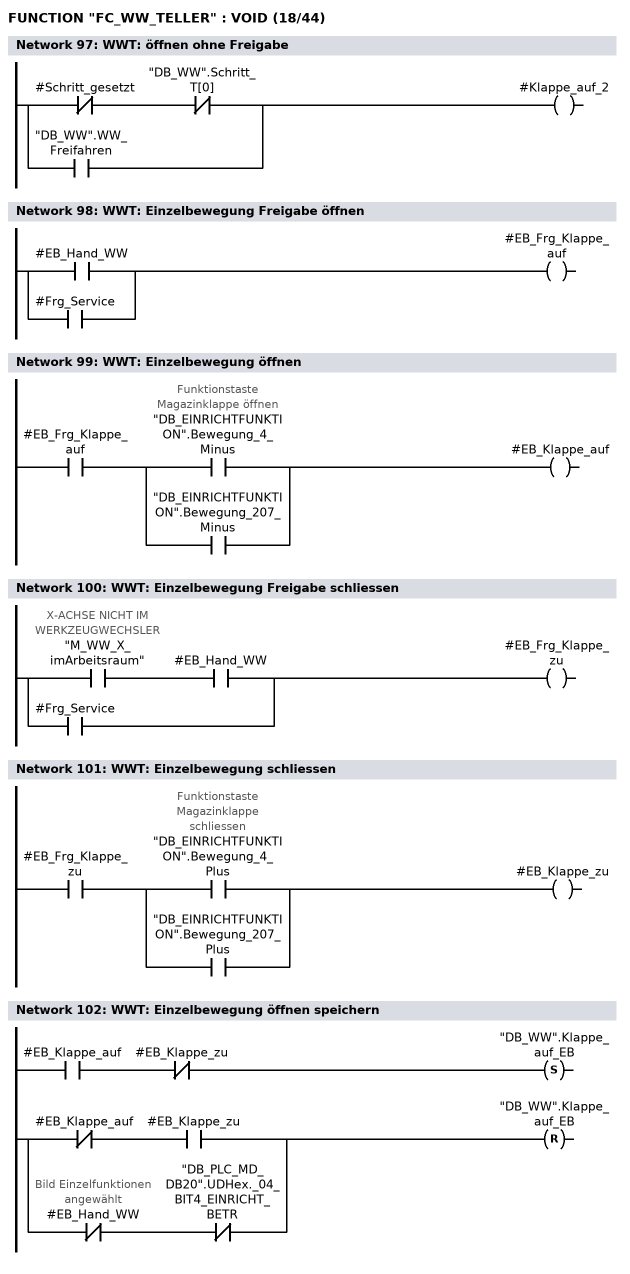

      UN    #Schritt_gesetzt;
      UN    "DB_WW".Schritt_T[0];
      O     "DB_WW".WW_Freifahren;
      =     #Klappe_auf_2;

NETWORK
TITLE =WWT: Einzelbewegung Freigabe öffnen

      O     #EB_Hand_WW;
      O     #Frg_Service;
      =     #EB_Frg_Klappe_auf;

NETWORK
TITLE =WWT: Einzelbewegung öffnen

      U     #EB_Frg_Klappe_auf;
      U(    ;
      O     "DB_EINRICHTFUNKTION".Bewegung_4_Minus; // Funktionstaste Magazinklappe öffnen
      O     "DB_EINRICHTFUNKTION".Bewegung_207_Minus;
      )     ;
      =     #EB_Klappe_auf;

NETWORK
TITLE =WWT: Einzelbewegung Freigabe schliessen

      U     "M_WW_X_imArbeitsraum"; // X-ACHSE NICHT IM WERKZEUGWECHSLER
      U     #EB_Hand_WW;
      O     #Frg_Service;
      =     #EB_Frg_Klappe_zu;

NETWORK
TITLE =WWT: Einzelbewegung schliessen

      U     #EB_Frg_Klappe_zu;
      U(    ;
      O     "DB_EINRICHTFUNKTION".Bewegung_4_Plus; // Funktionstaste Magazinklappe schliessen
      O     "DB_EINRICHTFUNKTION".Bewegung_207_Plus;
      )     ;
      =     #EB_Klappe_zu;

NETWORK
TITLE =WWT: Einzelbewegung öffnen speichern

      U     #EB_Klappe_auf;
      UN    #EB_Klappe_zu;
      S     "DB_WW".Klappe_auf_EB;

      U(    ;
      UN    #EB_Klappe_auf;
      U     #EB_Klappe_zu;
      O     ;
      UN    #EB_Hand_WW; // Bild Einzelfunktionen angewählt
      UN    "DB_PLC_MD_DB20".UDHex._04_BIT4_EINRICHT_BETR;
      )     ;
      R     "DB_WW".Klappe_auf_EB;
      NOP   0;

NETWORK
TITLE =WWT: Einzelbewegung schliessen speichern
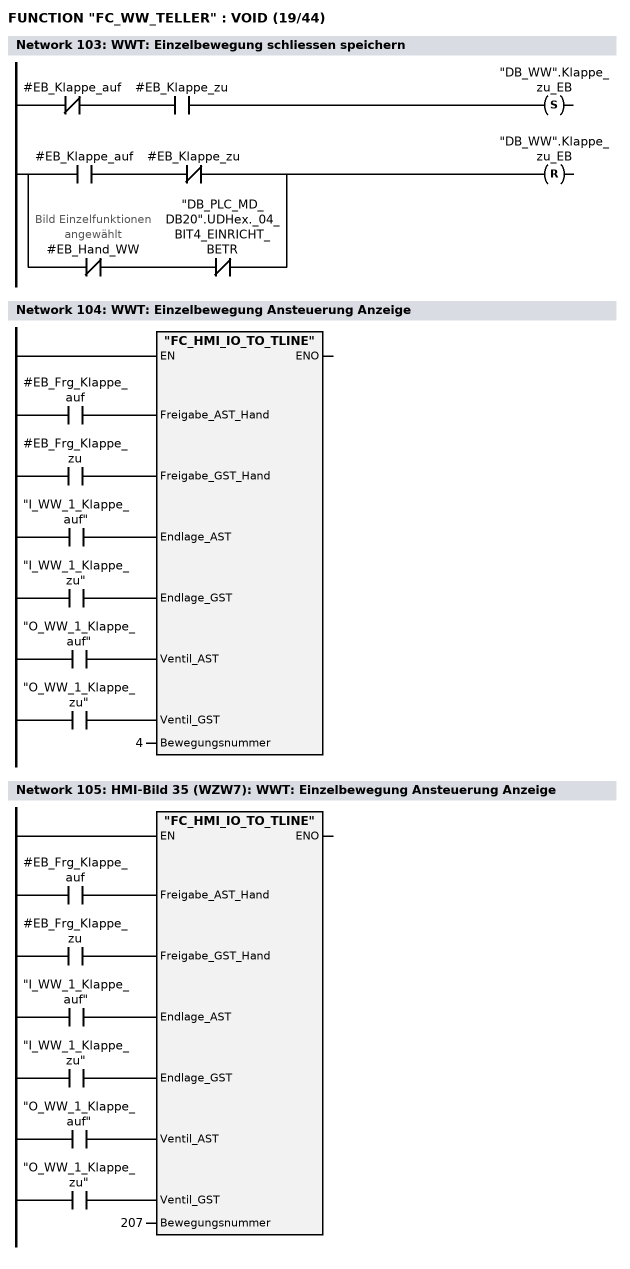

      UN    #EB_Klappe_auf;
      U     #EB_Klappe_zu;
      S     "DB_WW".Klappe_zu_EB;

      U(    ;
      U     #EB_Klappe_auf;
      UN    #EB_Klappe_zu;
      O     ;
      UN    #EB_Hand_WW; // Bild Einzelfunktionen angewählt
      UN    "DB_PLC_MD_DB20".UDHex._04_BIT4_EINRICHT_BETR;
      )     ;
      R     "DB_WW".Klappe_zu_EB;
      NOP   0;

NETWORK
TITLE =WWT: Einzelbewegung Ansteuerung Anzeige

      U     #EB_Frg_Klappe_auf;
      =     L     24.0;
      BLD   103;
      U     #EB_Frg_Klappe_zu;
      =     L     24.1;
      BLD   103;
      U     "I_WW_1_Klappe_auf";
      =     L     24.2;
      BLD   103;
      U     "I_WW_1_Klappe_zu";
      =     L     24.3;
      BLD   103;
      U     "O_WW_1_Klappe_auf";
      =     L     24.4;
      BLD   103;
      U     "O_WW_1_Klappe_zu";
      =     L     24.5;
      BLD   103;
      CALL "FC_HMI_IO_TO_TLINE" (
           Freigabe_AST_Hand        := L     24.0,
           Freigabe_GST_Hand        := L     24.1,
           Endlage_AST              := L     24.2,
           Endlage_GST              := L     24.3,
           Ventil_AST               := L     24.4,
           Ventil_GST               := L     24.5,
           Bewegungsnummer          := 4);
      NOP   0;
NETWORK
TITLE =HMI-Bild 35 (WZW7): WWT: Einzelbewegung Ansteuerung Anzeige

      U     #EB_Frg_Klappe_auf;
      =     L     24.0;
      BLD   103;
      U     #EB_Frg_Klappe_zu;
      =     L     24.1;
      BLD   103;
      U     "I_WW_1_Klappe_auf";
      =     L     24.2;
      BLD   103;
      U     "I_WW_1_Klappe_zu";
      =     L     24.3;
      BLD   103;
      U     "O_WW_1_Klappe_auf";
      =     L     24.4;
      BLD   103;
      U     "O_WW_1_Klappe_zu";
      =     L     24.5;
      BLD   103;
      CALL "FC_HMI_IO_TO_TLINE" (
           Freigabe_AST_Hand        := L     24.0,
           Freigabe_GST_Hand        := L     24.1,
           Endlage_AST              := L     24.2,
           Endlage_GST              := L     24.3,
           Ventil_AST               := L     24.4,
           Ventil_GST               := L     24.5,
           Bewegungsnummer          := 207);
      NOP   0;
NETWORK
TITLE =WWT: Ausgang öffnen
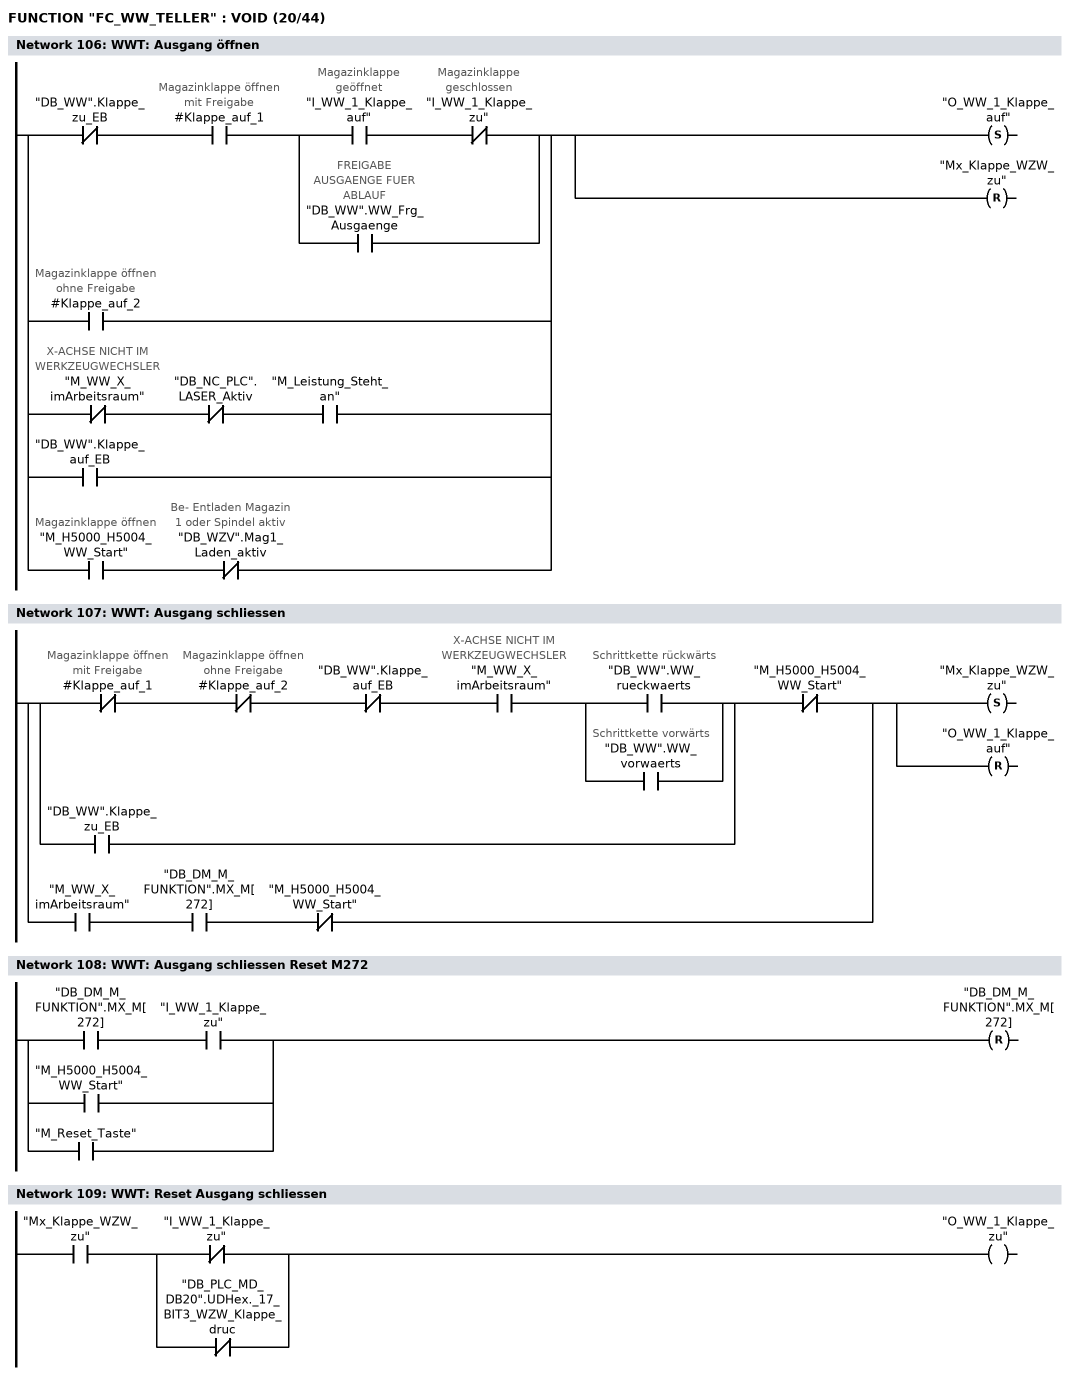

      UN    "DB_WW".Klappe_zu_EB;
      U     #Klappe_auf_1; // Magazinklappe öffnen mit Freigabe
      U(    ;
      U     "I_WW_1_Klappe_auf"; // Magazinklappe geöffnet
      UN    "I_WW_1_Klappe_zu"; // Magazinklappe geschlossen
      O     "DB_WW".WW_Frg_Ausgaenge; // FREIGABE AUSGAENGE FUER ABLAUF
      )     ;
      O     #Klappe_auf_2; // Magazinklappe öffnen ohne Freigabe
      O     ;
      UN    "M_WW_X_imArbeitsraum"; // X-ACHSE NICHT IM WERKZEUGWECHSLER
      UN    "DB_NC_PLC".LASER_Aktiv;
      U     "M_Leistung_Steht_an";
      O     "DB_WW".Klappe_auf_EB;
      O     ;
      U     "M_H5000_H5004_WW_Start"; // Magazinklappe öffnen
      UN    "DB_WZV".Mag1_Laden_aktiv; // Be- Entladen Magazin 1 oder Spindel aktiv
      S     "O_WW_1_Klappe_auf";

      R     "Mx_Klappe_WZW_zu";
NETWORK
TITLE =WWT: Ausgang schliessen

      U(    ;
      UN    #Klappe_auf_1; // Magazinklappe öffnen mit Freigabe
      UN    #Klappe_auf_2; // Magazinklappe öffnen ohne Freigabe
      UN    "DB_WW".Klappe_auf_EB;
      U     "M_WW_X_imArbeitsraum"; // X-ACHSE NICHT IM WERKZEUGWECHSLER
//      U     "I_WW_1_Klappe_zu"
      U(    ;
      O     "DB_WW".WW_rueckwaerts; // Schrittkette rückwärts
      O     "DB_WW".WW_vorwaerts; // Schrittkette vorwärts
      )     ;
      O     "DB_WW".Klappe_zu_EB;
      )     ;
      UN    "M_H5000_H5004_WW_Start";
      O     ;
      U     "M_WW_X_imArbeitsraum";
      U     "DB_DM_M_FUNKTION".MX_M[272];
      UN    "M_H5000_H5004_WW_Start";
      S     "Mx_Klappe_WZW_zu";
      R     "O_WW_1_Klappe_auf";

NETWORK
TITLE =WWT: Ausgang schliessen Reset M272

      U     "DB_DM_M_FUNKTION".MX_M[272];
      U     "I_WW_1_Klappe_zu";
      O     "M_H5000_H5004_WW_Start";
      O     "M_Reset_Taste";
      R     "DB_DM_M_FUNKTION".MX_M[272];

NETWORK
TITLE =WWT: Reset Ausgang schliessen

      U     "Mx_Klappe_WZW_zu";
      U(    ;
      ON    "I_WW_1_Klappe_zu";
      ON    "DB_PLC_MD_DB20".UDHex._17_BIT3_WZW_Klappe_druc;
      )     ;
      =     "O_WW_1_Klappe_zu";

NETWORK
TITLE =========== Werkzeug in / aus Spindel ===============



NETWORK
TITLE =WZHUB: BEFEHL FAHRE auf AUSFAHRPOSITION
// AUS DEN SCHRITTMERKERN WERDEN VERSCHIEDENE BEFEHLE ERZEUGT, DIE
// WIEDERUM VERSCHIEDENE AKTION AUSLOESEN.
//
// BEFEHL FAHRE Z-Achse auf AUSFAHRPOSITION
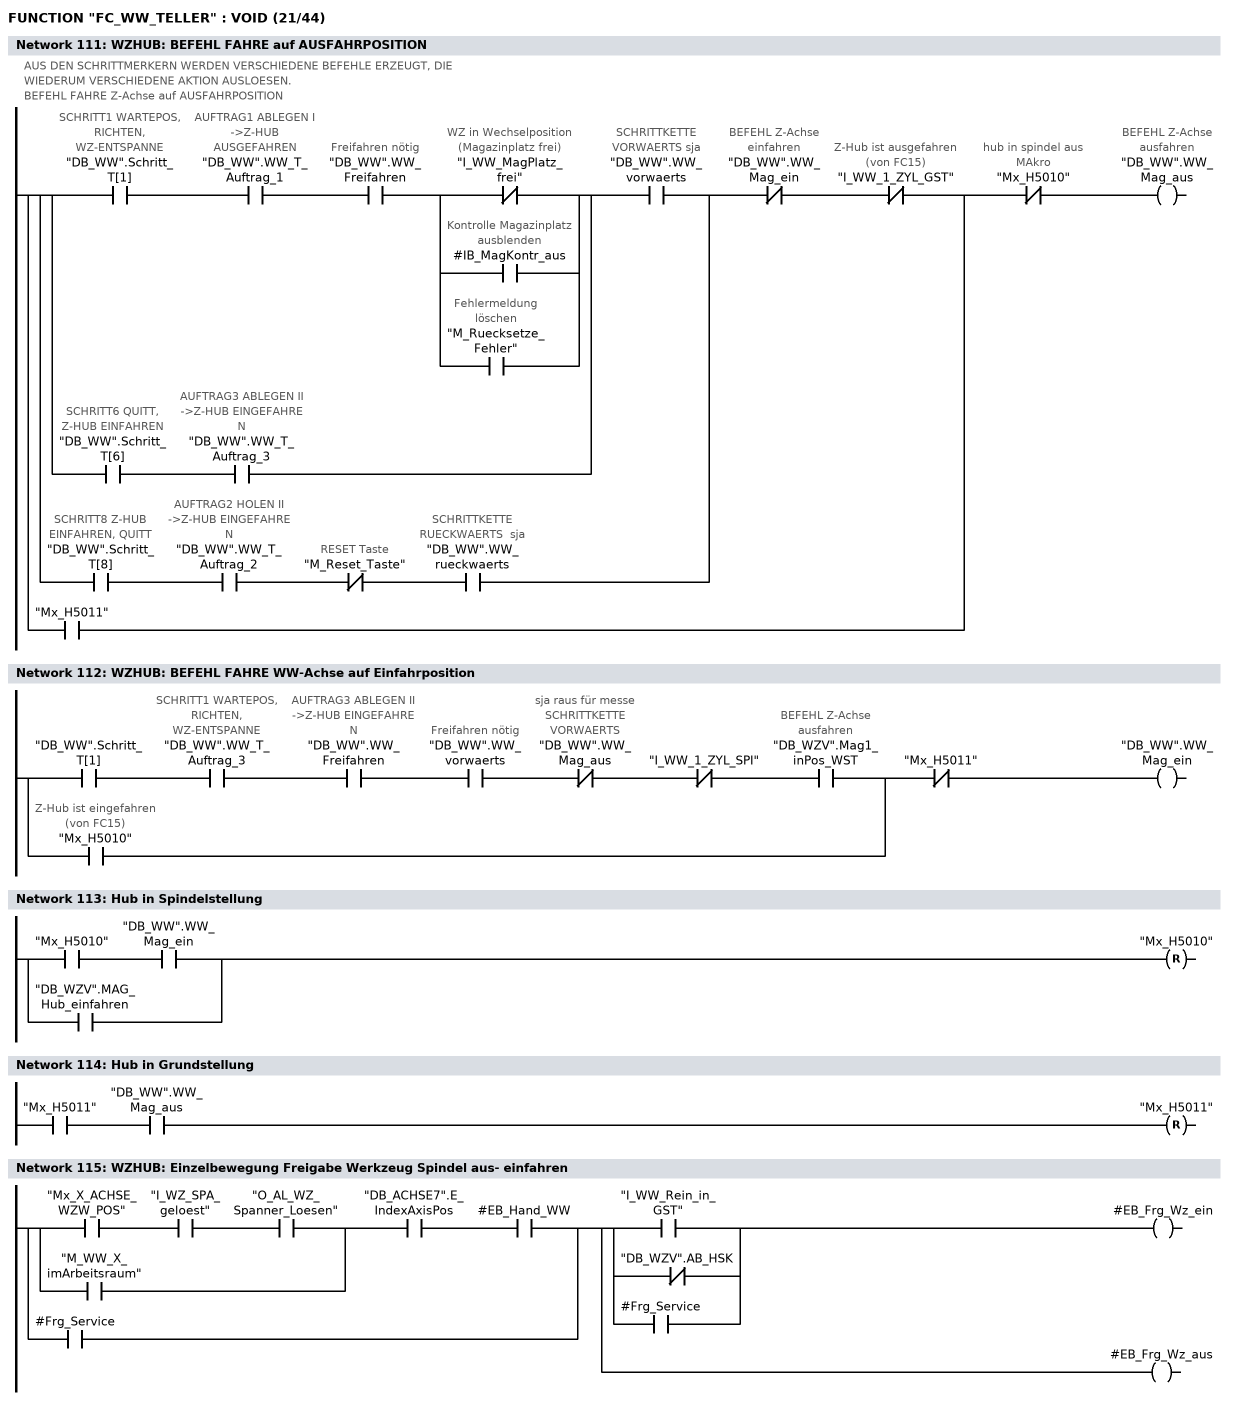
      U(    ;
      U(    ;
      U(    ;
      U     "DB_WW".Schritt_T[1]; // SCHRITT1 WARTEPOS, RICHTEN, WZ-ENTSPANNE
      U     "DB_WW".WW_T_Auftrag_1; // AUFTRAG1 ABLEGEN I ->Z-HUB AUSGEFAHREN
      U     "DB_WW".WW_Freifahren; // Freifahren nötig
      U(    ;
      ON    "I_WW_MagPlatz_frei"; // WZ in Wechselposition (Magazinplatz frei)
      O     #IB_MagKontr_aus; // Kontrolle Magazinplatz ausblenden
      O     "M_Ruecksetze_Fehler"; // Fehlermeldung löschen
      )     ;
      O     ;
      U     "DB_WW".Schritt_T[6]; // SCHRITT6 QUITT, Z-HUB EINFAHREN
      U     "DB_WW".WW_T_Auftrag_3; // AUFTRAG3 ABLEGEN II ->Z-HUB EINGEFAHREN
      )     ;
      U     "DB_WW".WW_vorwaerts; // SCHRITTKETTE VORWAERTS sja
      O     ;
      U     "DB_WW".Schritt_T[8]; // SCHRITT8 Z-HUB EINFAHREN, QUITT
      U     "DB_WW".WW_T_Auftrag_2; // AUFTRAG2 HOLEN II ->Z-HUB EINGEFAHREN
      UN    "M_Reset_Taste"; // RESET Taste
      U     "DB_WW".WW_rueckwaerts; // SCHRITTKETTE RUECKWAERTS  sja
      )     ;
      UN    "DB_WW".WW_Mag_ein; // BEFEHL Z-Achse einfahren
      UN    "I_WW_1_ZYL_GST"; // Z-Hub ist ausgefahren (von FC15)
      O     "Mx_H5011";
      )     ;
      UN    "Mx_H5010"; // hub in spindel aus MAkro
      =     "DB_WW".WW_Mag_aus; // BEFEHL Z-Achse ausfahren

NETWORK
TITLE =WZHUB: BEFEHL FAHRE WW-Achse auf Einfahrposition

      U(    ;
      U     "DB_WW".Schritt_T[1];
      U     "DB_WW".WW_T_Auftrag_3; // SCHRITT1 WARTEPOS, RICHTEN, WZ-ENTSPANNE
      U     "DB_WW".WW_Freifahren; // AUFTRAG3 ABLEGEN II ->Z-HUB EINGEFAHREN
      U     "DB_WW".WW_vorwaerts; // Freifahren nötig
      UN    "DB_WW".WW_Mag_aus; //sja raus für messe SCHRITTKETTE VORWAERTS
//      O
//      U     "DB_WW".Schritt_T[1]        // SCHRITT1 WARTEPOS, RICHTEN, WZ-ENTSPANNE
//      U     "DB_WW".WW_T_Auftrag_1      // AUFTRAG1 ABLEGEN I ->Z-HUB AUSGEFAHREN
//      UN    "M_Reset_Taste"             // RESET Taste
//      U     "DB_WW".WW_rueckwaerts      // sja raus für messe SCHRITTKETTE RUECKWAERTS
      UN    "I_WW_1_ZYL_SPI";
      U     "DB_WZV".Mag1_inPos_WST; // BEFEHL Z-Achse ausfahren
      O     "Mx_H5010"; // Z-Hub ist eingefahren (von FC15)
      )     ;
      UN    "Mx_H5011";
      =     "DB_WW".WW_Mag_ein;
NETWORK
TITLE =Hub in Spindelstellung

      U     "Mx_H5010";
      U     "DB_WW".WW_Mag_ein;
      O     "DB_WZV".MAG_Hub_einfahren;
      R     "Mx_H5010";
NETWORK
TITLE =Hub in Grundstellung

      U     "Mx_H5011";
      U     "DB_WW".WW_Mag_aus;
      R     "Mx_H5011";
NETWORK
TITLE =WZHUB: Einzelbewegung Freigabe Werkzeug Spindel aus- einfahren

      U(    ;
      U     "Mx_X_ACHSE_WZW_POS";
      U     "I_WZ_SPA_geloest";
      U     "O_AL_WZ_Spanner_Loesen";
      O     "M_WW_X_imArbeitsraum";
      )     ;
      U     "DB_ACHSE7".E_IndexAxisPos;
      U     #EB_Hand_WW;
      O     #Frg_Service;
      =     L     24.0;
      U     L     24.0;
      U(    ;
      O     "I_WW_Rein_in_GST";
      ON    "DB_WZV".AB_HSK;
      O     #Frg_Service;
      )     ;
      =     #EB_Frg_Wz_ein;
      U     L     24.0;
      BLD   102;
      =     #EB_Frg_Wz_aus;
NETWORK
TITLE =WZHUB: Einzelbewegung Werkzeug aus Spindel ausfahren
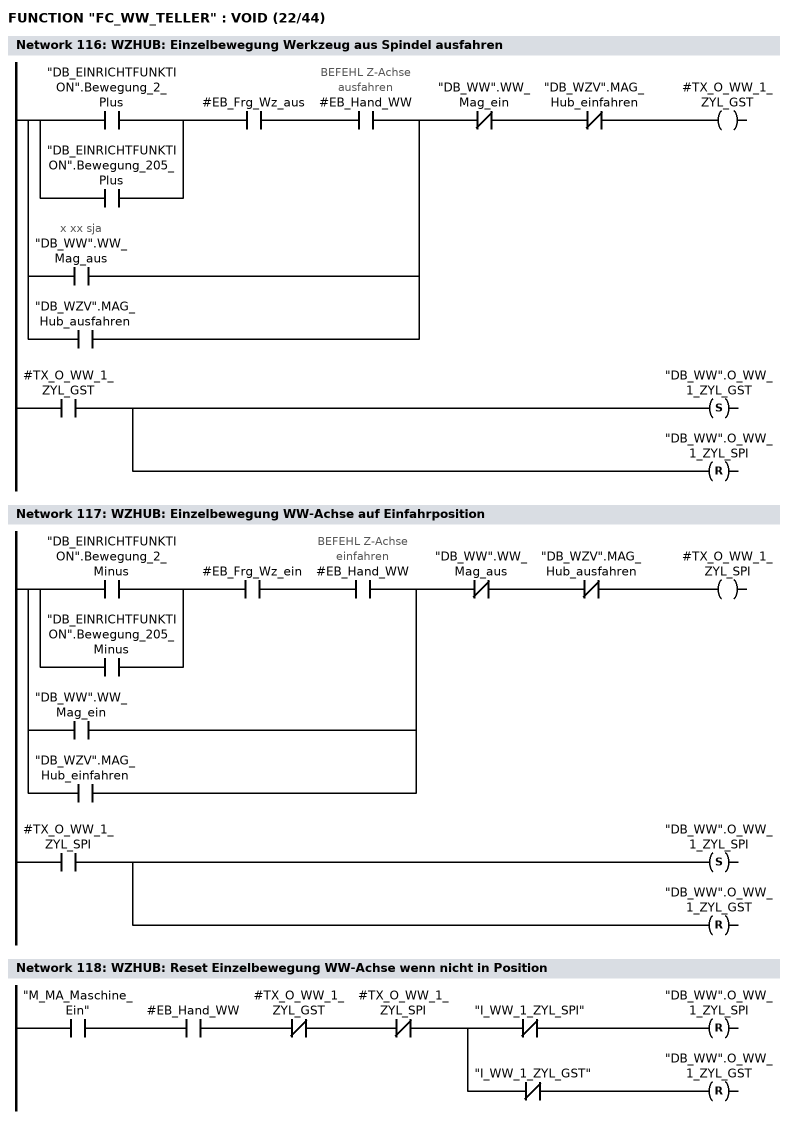

      U(    ;
      U(    ;
      O     "DB_EINRICHTFUNKTION".Bewegung_2_Plus;
      O     "DB_EINRICHTFUNKTION".Bewegung_205_Plus;
      )     ;
      U     #EB_Frg_Wz_aus;
      U     #EB_Hand_WW; // BEFEHL Z-Achse ausfahren
//      O     "DB_WZV".MAG_Hub_einfahren  // xxx sja
      O     "DB_WW".WW_Mag_aus; // x xx sja
      O     "DB_WZV".MAG_Hub_ausfahren;
      )     ;
// =     "DB_WW".ASUP_Rettung.WW_Hub_ausfahren

      UN    "DB_WW".WW_Mag_ein;
      UN    "DB_WZV".MAG_Hub_einfahren;
      =     #TX_O_WW_1_ZYL_GST;
      U     #TX_O_WW_1_ZYL_GST;
      S     "DB_WW".O_WW_1_ZYL_GST;
      R     "DB_WW".O_WW_1_ZYL_SPI;
NETWORK
TITLE =WZHUB: Einzelbewegung WW-Achse auf Einfahrposition

      U(    ;
      U(    ;
      O     "DB_EINRICHTFUNKTION".Bewegung_2_Minus;
      O     "DB_EINRICHTFUNKTION".Bewegung_205_Minus;
      )     ;
      U     #EB_Frg_Wz_ein;
      U     #EB_Hand_WW; // BEFEHL Z-Achse einfahren
      O     "DB_WW".WW_Mag_ein;
      O     "DB_WZV".MAG_Hub_einfahren;
      )     ;

// =     "DB_WW".ASUP_Rettung.WW_Hub_einfahren

      UN    "DB_WW".WW_Mag_aus;
      UN    "DB_WZV".MAG_Hub_ausfahren;
      =     #TX_O_WW_1_ZYL_SPI;
      U     #TX_O_WW_1_ZYL_SPI;
      S     "DB_WW".O_WW_1_ZYL_SPI;
      R     "DB_WW".O_WW_1_ZYL_GST;
NETWORK
TITLE =WZHUB: Reset Einzelbewegung WW-Achse wenn nicht in Position

      U     "M_MA_Maschine_Ein";
      U     #EB_Hand_WW;
      UN    #TX_O_WW_1_ZYL_GST;
      UN    #TX_O_WW_1_ZYL_SPI;
      =     L     24.0;
      U     L     24.0;
      UN    "I_WW_1_ZYL_SPI";
      R     "DB_WW".O_WW_1_ZYL_SPI;
      U     L     24.0;
      UN    "I_WW_1_ZYL_GST";
      R     "DB_WW".O_WW_1_ZYL_GST;
NETWORK
TITLE =WZHUB: Freigabe Ansteuerung Ventil Hub ein- / ausfahren
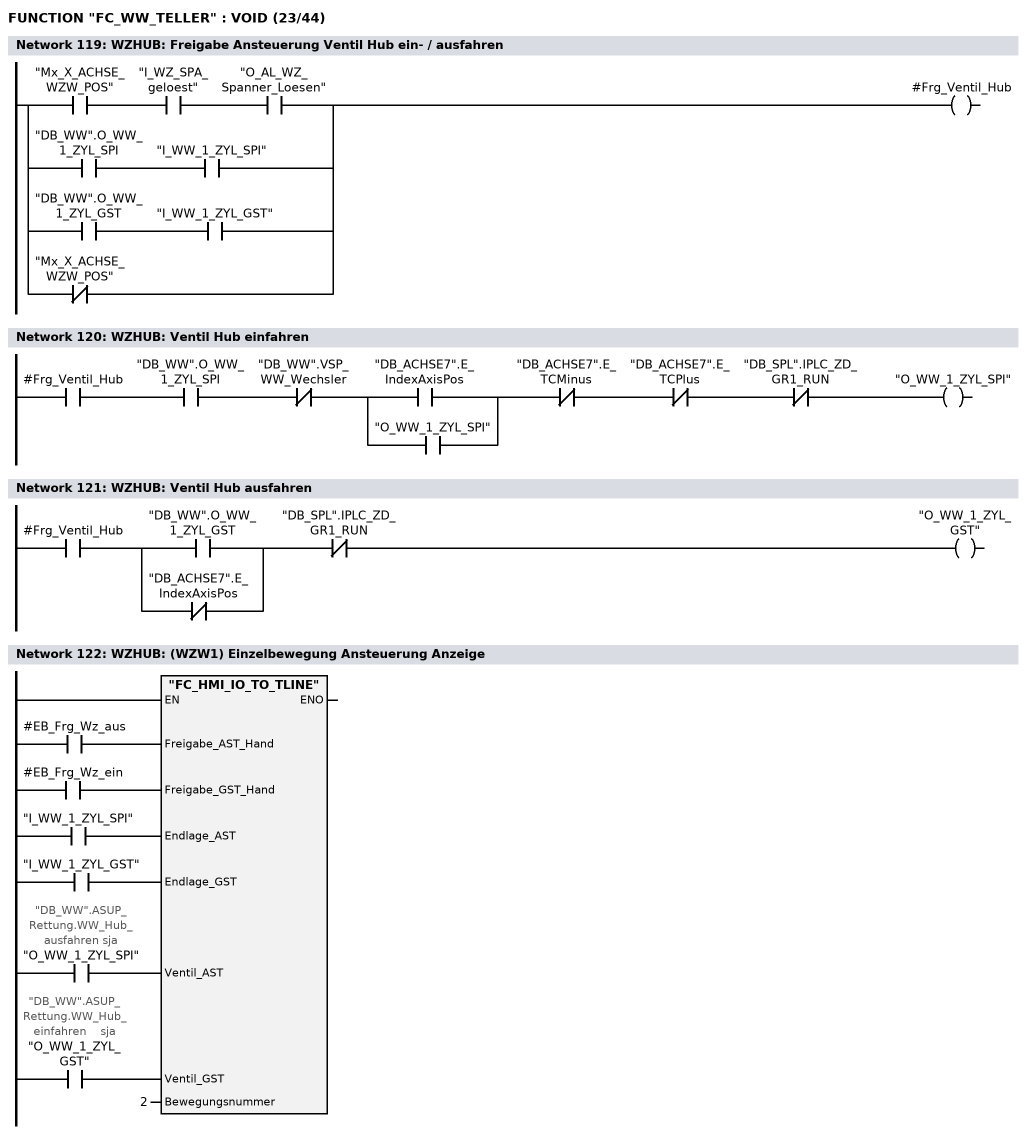

      U     "Mx_X_ACHSE_WZW_POS";
      U     "I_WZ_SPA_geloest";
      U     "O_AL_WZ_Spanner_Loesen";
      O     ;
      U     "DB_WW".O_WW_1_ZYL_SPI;
      U     "I_WW_1_ZYL_SPI";
      O     ;
      U     "DB_WW".O_WW_1_ZYL_GST;
      U     "I_WW_1_ZYL_GST";
      ON    "Mx_X_ACHSE_WZW_POS";
      =     #Frg_Ventil_Hub;

NETWORK
TITLE =WZHUB: Ventil Hub einfahren

      U     #Frg_Ventil_Hub;
      U     "DB_WW".O_WW_1_ZYL_SPI;
      UN    "DB_WW".VSP_WW_Wechsler;
      U(    ;
      O     "DB_ACHSE7".E_IndexAxisPos;
      O     "O_WW_1_ZYL_SPI";
      )     ;

      UN    "DB_ACHSE7".E_TCMinus;
      UN    "DB_ACHSE7".E_TCPlus;
      UN    "DB_SPL".IPLC_ZD_GR1_RUN;
      =     "O_WW_1_ZYL_SPI";
NETWORK
TITLE =WZHUB: Ventil Hub ausfahren

      U     #Frg_Ventil_Hub;
      U(    ;
      O     "DB_WW".O_WW_1_ZYL_GST;
      ON    "DB_ACHSE7".E_IndexAxisPos;
      )     ;
      UN    "DB_SPL".IPLC_ZD_GR1_RUN;

      =     "O_WW_1_ZYL_GST";
NETWORK
TITLE =WZHUB: (WZW1) Einzelbewegung Ansteuerung Anzeige

      U     #EB_Frg_Wz_aus;
      =     L     24.0;
      BLD   103;
      U     #EB_Frg_Wz_ein;
      =     L     24.1;
      BLD   103;
      U     "I_WW_1_ZYL_SPI";
      =     L     24.2;
      BLD   103;
      U     "I_WW_1_ZYL_GST";
      =     L     24.3;
      BLD   103;
      U     "O_WW_1_ZYL_SPI"; //"DB_WW".ASUP_Rettung.WW_Hub_ausfahren sja
      =     L     24.4;
      BLD   103;
      U     "O_WW_1_ZYL_GST"; //"DB_WW".ASUP_Rettung.WW_Hub_einfahren    sja
      =     L     24.5;
      BLD   103;
      CALL "FC_HMI_IO_TO_TLINE" (
           Freigabe_AST_Hand        := L     24.0,
           Freigabe_GST_Hand        := L     24.1,
           Endlage_AST              := L     24.2,
           Endlage_GST              := L     24.3,
           Ventil_AST               := L     24.4,
           Ventil_GST               := L     24.5,
           Bewegungsnummer          := 2);
      NOP   0;
NETWORK
TITLE =WZHUB: (WZW7) Einzelbewegung Ansteuerung Anzeige
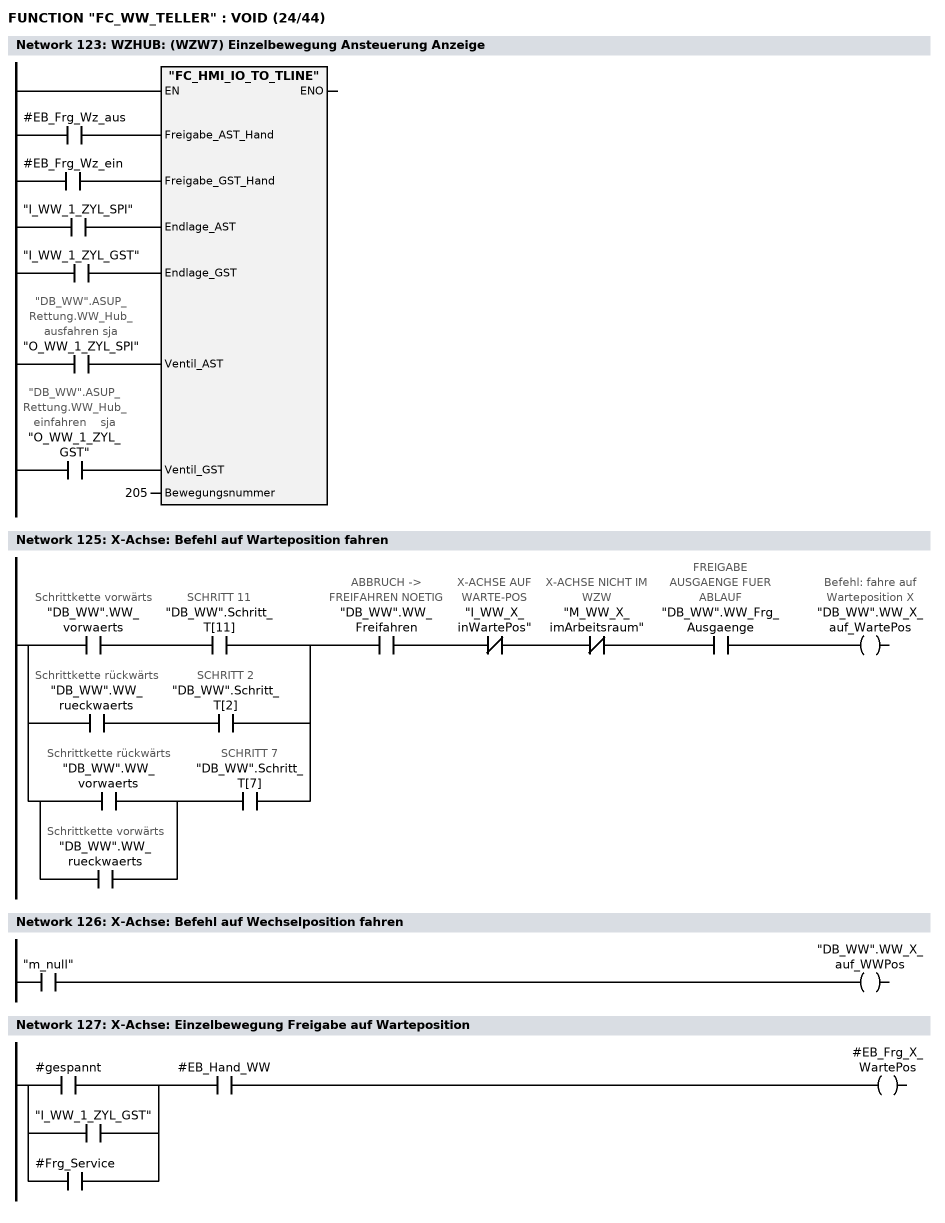

      U     #EB_Frg_Wz_aus;
      =     L     24.0;
      BLD   103;
      U     #EB_Frg_Wz_ein;
      =     L     24.1;
      BLD   103;
      U     "I_WW_1_ZYL_SPI";
      =     L     24.2;
      BLD   103;
      U     "I_WW_1_ZYL_GST";
      =     L     24.3;
      BLD   103;
      U     "O_WW_1_ZYL_SPI"; //"DB_WW".ASUP_Rettung.WW_Hub_ausfahren sja
      =     L     24.4;
      BLD   103;
      U     "O_WW_1_ZYL_GST"; //"DB_WW".ASUP_Rettung.WW_Hub_einfahren    sja
      =     L     24.5;
      BLD   103;
      CALL "FC_HMI_IO_TO_TLINE" (
           Freigabe_AST_Hand        := L     24.0,
           Freigabe_GST_Hand        := L     24.1,
           Endlage_AST              := L     24.2,
           Endlage_GST              := L     24.3,
           Ventil_AST               := L     24.4,
           Ventil_GST               := L     24.5,
           Bewegungsnummer          := 205);
      NOP   0;
NETWORK
TITLE ============ Spindel in / aus Werkzeugwechsler ============



NETWORK
TITLE =X-Achse: Befehl auf Warteposition fahren

      U(    ;
      U     "DB_WW".WW_vorwaerts; // Schrittkette vorwärts
      U     "DB_WW".Schritt_T[11]; // SCHRITT 11
      O     ;
      U     "DB_WW".WW_rueckwaerts; // Schrittkette rückwärts
      U     "DB_WW".Schritt_T[2]; // SCHRITT 2
      O     ;
      U(    ;
      O     "DB_WW".WW_vorwaerts; // Schrittkette rückwärts
      O     "DB_WW".WW_rueckwaerts; // Schrittkette vorwärts
      )     ;
      U     "DB_WW".Schritt_T[7]; // SCHRITT 7
      )     ;
      U     "DB_WW".WW_Freifahren; // ABBRUCH -> FREIFAHREN NOETIG
      UN    "I_WW_X_inWartePos"; // X-ACHSE AUF WARTE-POS
      UN    "M_WW_X_imArbeitsraum"; // X-ACHSE NICHT IM WZW
      U     "DB_WW".WW_Frg_Ausgaenge; // FREIGABE AUSGAENGE FUER ABLAUF
      =     "DB_WW".WW_X_auf_WartePos; // Befehl: fahre auf Warteposition X

NETWORK
TITLE =X-Achse: Befehl auf Wechselposition fahren

      U     "m_null";
      =     "DB_WW".WW_X_auf_WWPos;

NETWORK
TITLE =X-Achse: Einzelbewegung Freigabe auf Warteposition

      U(    ;
      O     #gespannt;
      O     "I_WW_1_ZYL_GST";
      O     #Frg_Service;

      )     ;
      U     #EB_Hand_WW;
      =     #EB_Frg_X_WartePos;
NETWORK
TITLE =X-Achse: Einzelbewegung auf Warteposition fahren
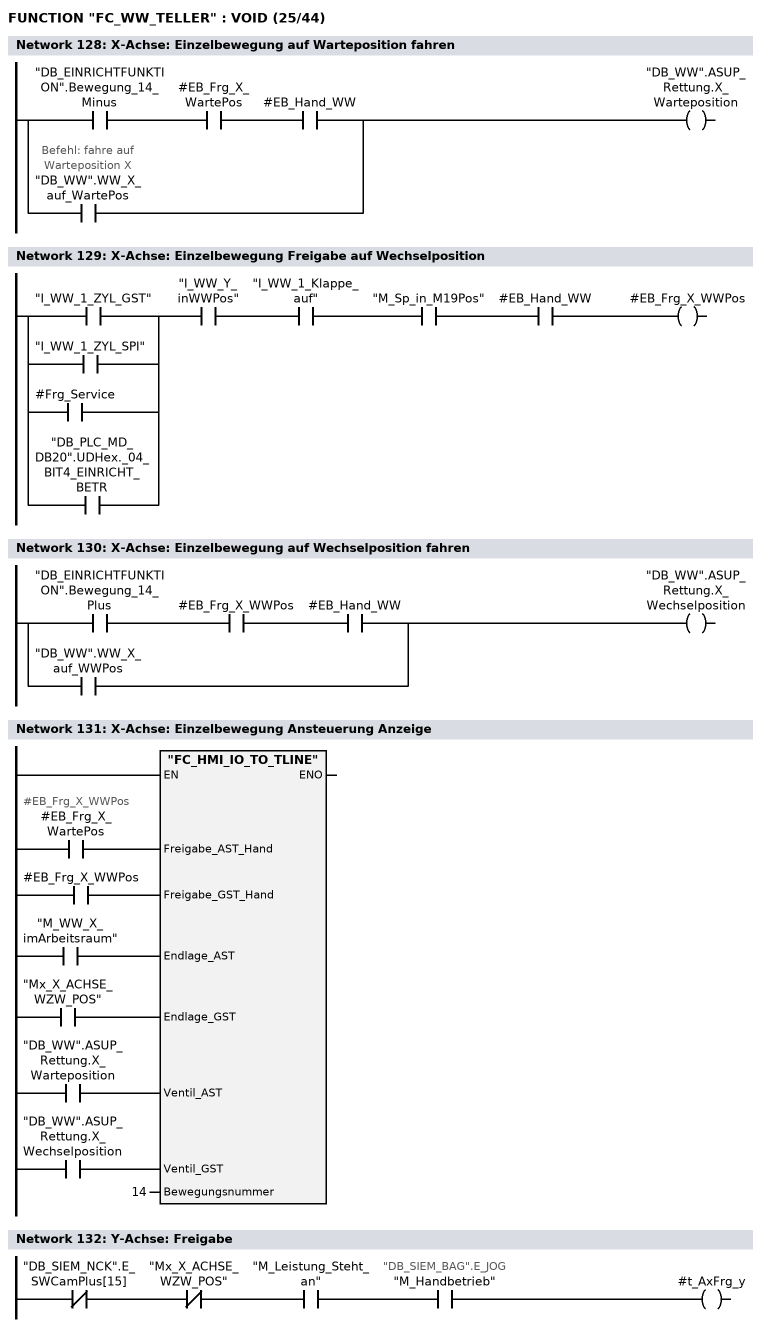

      U     "DB_EINRICHTFUNKTION".Bewegung_14_Minus;
      U     #EB_Frg_X_WartePos;
      U     #EB_Hand_WW;
      O     "DB_WW".WW_X_auf_WartePos; // Befehl: fahre auf Warteposition X
      =     "DB_WW".ASUP_Rettung.X_Warteposition;

NETWORK
TITLE =X-Achse: Einzelbewegung Freigabe auf Wechselposition

      U(    ;
      O     "I_WW_1_ZYL_GST";
      O     "I_WW_1_ZYL_SPI";
      O     #Frg_Service;
      O     "DB_PLC_MD_DB20".UDHex._04_BIT4_EINRICHT_BETR;
      )     ;
      U     "I_WW_Y_inWWPos";
      U     "I_WW_1_Klappe_auf";

      U     "M_Sp_in_M19Pos";
      U     #EB_Hand_WW;
      =     #EB_Frg_X_WWPos;
NETWORK
TITLE =X-Achse: Einzelbewegung auf Wechselposition fahren

      U     "DB_EINRICHTFUNKTION".Bewegung_14_Plus;
      U     #EB_Frg_X_WWPos;
      U     #EB_Hand_WW;
      O     "DB_WW".WW_X_auf_WWPos;
      =     "DB_WW".ASUP_Rettung.X_Wechselposition;

NETWORK
TITLE =X-Achse: Einzelbewegung Ansteuerung Anzeige

      U     #EB_Frg_X_WartePos; //#EB_Frg_X_WWPos
      =     L     24.0;
      BLD   103;
      U     #EB_Frg_X_WWPos;
      =     L     24.1;
      BLD   103;
      U     "M_WW_X_imArbeitsraum";
      =     L     24.2;
      BLD   103;
      U     "Mx_X_ACHSE_WZW_POS";
      =     L     24.3;
      BLD   103;
      U     "DB_WW".ASUP_Rettung.X_Warteposition;
      =     L     24.4;
      BLD   103;
      U     "DB_WW".ASUP_Rettung.X_Wechselposition;
      =     L     24.5;
      BLD   103;
      CALL "FC_HMI_IO_TO_TLINE" (
           Freigabe_AST_Hand        := L     24.0,
           Freigabe_GST_Hand        := L     24.1,
           Endlage_AST              := L     24.2,
           Endlage_GST              := L     24.3,
           Ventil_AST               := L     24.4,
           Ventil_GST               := L     24.5,
           Bewegungsnummer          := 14);//176
      NOP   0;
NETWORK
TITLE =Y-Achse: Freigabe

      UN    "DB_SIEM_NCK".E_SWCamPlus[15];
      UN    "Mx_X_ACHSE_WZW_POS";
      U     "M_Leistung_Steht_an";
      U     "M_Handbetrieb"; // "DB_SIEM_BAG".E_JOG
      =     #t_AxFrg_y;

NETWORK
TITLE =Y-Achse: Fahrbefehl
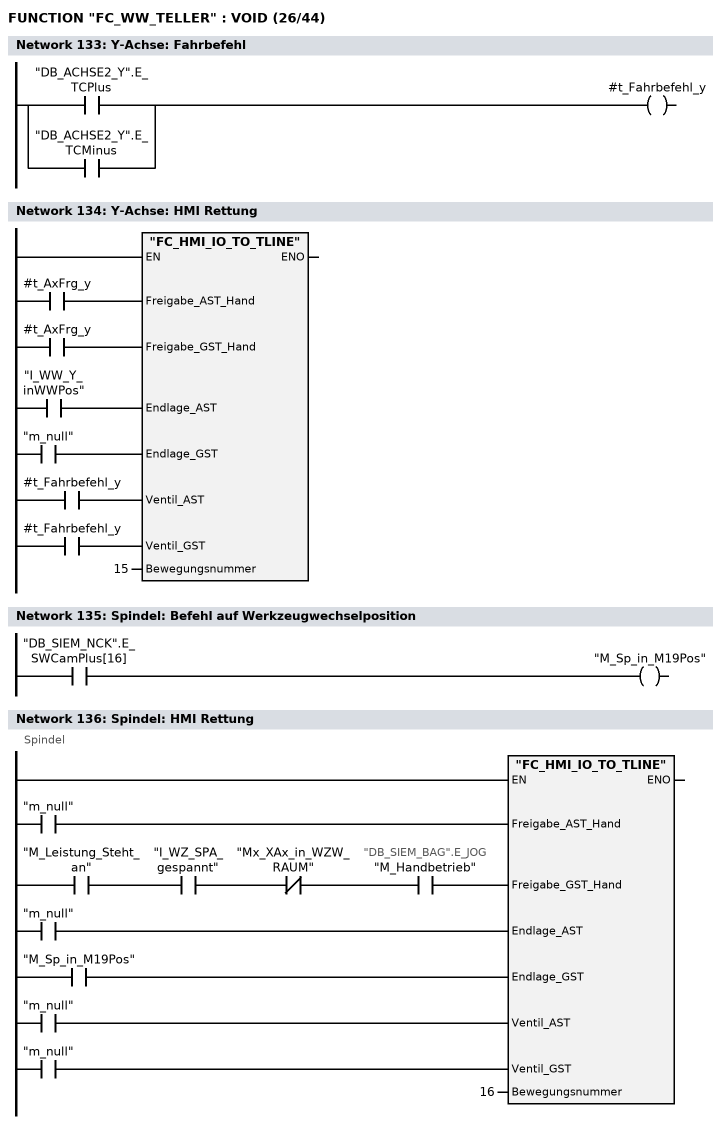

      O     "DB_ACHSE2_Y".E_TCPlus;
      O     "DB_ACHSE2_Y".E_TCMinus;
      =     #t_Fahrbefehl_y;
NETWORK
TITLE =Y-Achse: HMI Rettung
//
//
      U     #t_AxFrg_y;
      =     L     24.0;
      BLD   103;
      U     #t_AxFrg_y;
      =     L     24.1;
      BLD   103;
      U     "I_WW_Y_inWWPos";
      =     L     24.2;
      BLD   103;
      U     "m_null";
      =     L     24.3;
      BLD   103;
      U     #t_Fahrbefehl_y;
      =     L     24.4;
      BLD   103;
      U     #t_Fahrbefehl_y;
      =     L     24.5;
      BLD   103;
      CALL "FC_HMI_IO_TO_TLINE" (
           Freigabe_AST_Hand        := L     24.0,
           Freigabe_GST_Hand        := L     24.1,
           Endlage_AST              := L     24.2,
           Endlage_GST              := L     24.3,
           Ventil_AST               := L     24.4,
           Ventil_GST               := L     24.5,
           Bewegungsnummer          := 15);
      NOP   0;
NETWORK
TITLE =Spindel: Befehl auf Werkzeugwechselposition

      U     "DB_SIEM_NCK".E_SWCamPlus[16];
      =     "M_Sp_in_M19Pos";

NETWORK
TITLE =Spindel: HMI Rettung
//Spindel
      U     "m_null";
      =     L     24.0;
      BLD   103;
      U     "M_Leistung_Steht_an";
      U     "I_WZ_SPA_gespannt";
      UN    "Mx_XAx_in_WZW_RAUM";
      U     "M_Handbetrieb"; // "DB_SIEM_BAG".E_JOG
      =     L     24.1;
      BLD   103;
      U     "m_null";
      =     L     24.2;
      BLD   103;
      U     "M_Sp_in_M19Pos";
      =     L     24.3;
      BLD   103;
      U     "m_null";
      =     L     24.4;
      BLD   103;
      U     "m_null";
      =     L     24.5;
      BLD   103;
      CALL "FC_HMI_IO_TO_TLINE" (
           Freigabe_AST_Hand        := L     24.0,
           Freigabe_GST_Hand        := L     24.1,
           Endlage_AST              := L     24.2,
           Endlage_GST              := L     24.3,
           Ventil_AST               := L     24.4,
           Ventil_GST               := L     24.5,
           Bewegungsnummer          := 16);
      NOP   0;
NETWORK
TITLE ========= Werkzeug im Magazin entsichern Wechselstelle ========



NETWORK
TITLE =WW_MagTasche: BEFEHL Werkzeug entsichern Spindelseite
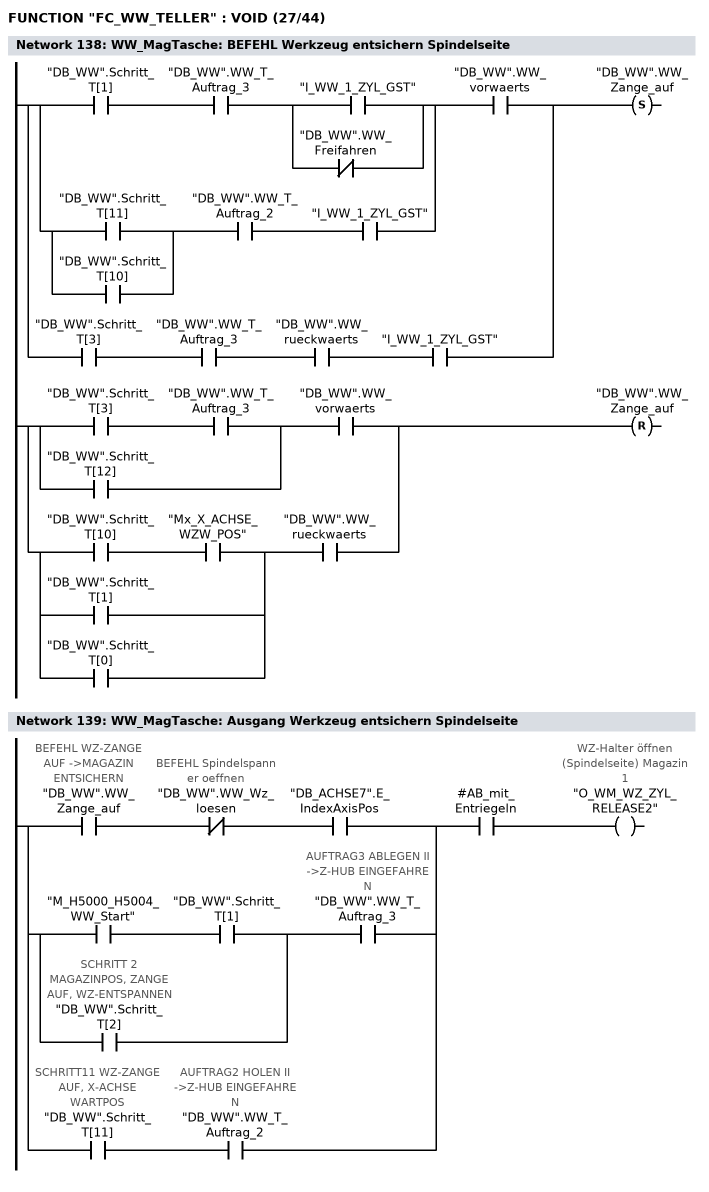

      U(    ;
      U(    ;
      U     "DB_WW".Schritt_T[1];
      U     "DB_WW".WW_T_Auftrag_3;
      U(    ;
      O     "I_WW_1_ZYL_GST";
      ON    "DB_WW".WW_Freifahren;
      )     ;
      O     ;
      U(    ;
      O     "DB_WW".Schritt_T[11];
      O     "DB_WW".Schritt_T[10];
      )     ;
      U     "DB_WW".WW_T_Auftrag_2;
      U     "I_WW_1_ZYL_GST";
      )     ;
      U     "DB_WW".WW_vorwaerts;
      O     ;
      U     "DB_WW".Schritt_T[3];
      U     "DB_WW".WW_T_Auftrag_3;
      U     "DB_WW".WW_rueckwaerts;
      U     "I_WW_1_ZYL_GST";

      )     ;
      S     "DB_WW".WW_Zange_auf;
      U(    ;
      U(    ;
      U     "DB_WW".Schritt_T[3];
      U     "DB_WW".WW_T_Auftrag_3;
      O     "DB_WW".Schritt_T[12];
      )     ;
      U     "DB_WW".WW_vorwaerts;
      O     ;
      U(    ;
      U     "DB_WW".Schritt_T[10];
      U     "Mx_X_ACHSE_WZW_POS";
      O     "DB_WW".Schritt_T[1];
      O     "DB_WW".Schritt_T[0];
      )     ;

      U     "DB_WW".WW_rueckwaerts;
      )     ;
      R     "DB_WW".WW_Zange_auf;
      NOP   0;
NETWORK
TITLE =WW_MagTasche: Ausgang Werkzeug entsichern Spindelseite

      U(    ;
      U     "DB_WW".WW_Zange_auf; // BEFEHL WZ-ZANGE AUF ->MAGAZIN ENTSICHERN
      UN    "DB_WW".WW_Wz_loesen; // BEFEHL Spindelspanner oeffnen
      U     "DB_ACHSE7".E_IndexAxisPos;
      O     ;
      U(    ;
      U     "M_H5000_H5004_WW_Start";
      U     "DB_WW".Schritt_T[1];
      O     "DB_WW".Schritt_T[2]; // SCHRITT 2 MAGAZINPOS, ZANGE AUF, WZ-ENTSPANNEN
      )     ;
      U     "DB_WW".WW_T_Auftrag_3; // AUFTRAG3 ABLEGEN II ->Z-HUB EINGEFAHREN
      O     ;
      U     "DB_WW".Schritt_T[11]; // SCHRITT11 WZ-ZANGE AUF, X-ACHSE WARTPOS
      U     "DB_WW".WW_T_Auftrag_2; // AUFTRAG2 HOLEN II ->Z-HUB EINGEFAHREN
      )     ;
      U     #AB_mit_Entriegeln;
      =     "O_WM_WZ_ZYL_RELEASE2"; // WZ-Halter öffnen (Spindelseite) Magazin 1

NETWORK
TITLE ========= Werkzeug im Magazin entsichern Ladestelle ========



NETWORK
TITLE =WM_MagTasche: Ausgang Werkzeug entsichern an BELADESTATION
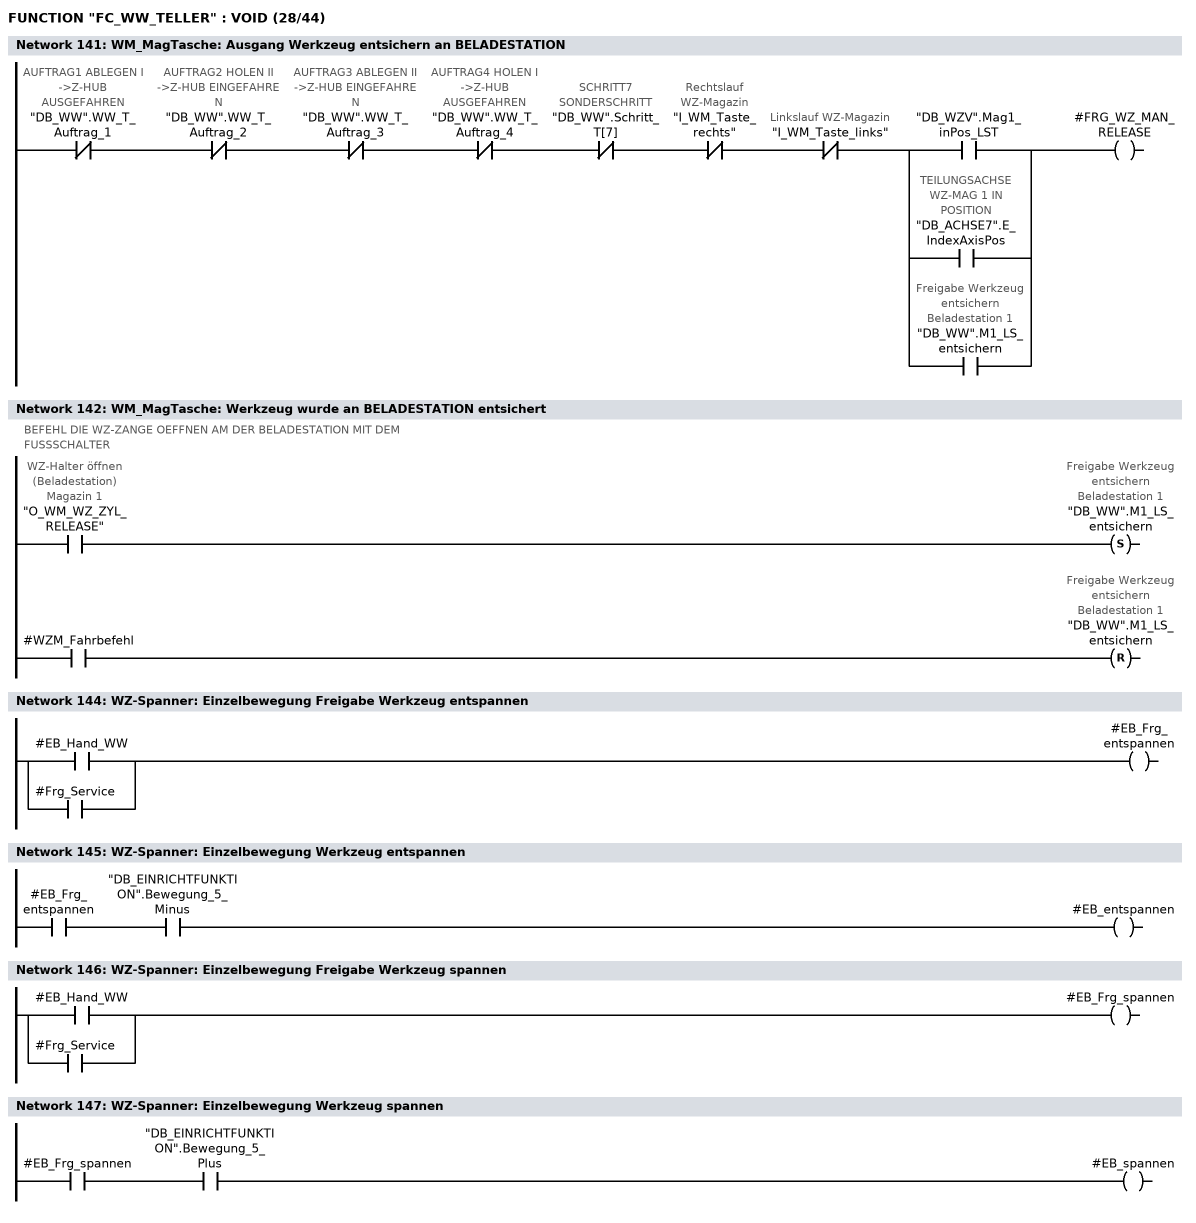

      UN    "DB_WW".WW_T_Auftrag_1; // AUFTRAG1 ABLEGEN I ->Z-HUB AUSGEFAHREN
      UN    "DB_WW".WW_T_Auftrag_2; // AUFTRAG2 HOLEN II ->Z-HUB EINGEFAHREN
      UN    "DB_WW".WW_T_Auftrag_3; // AUFTRAG3 ABLEGEN II ->Z-HUB EINGEFAHREN
      UN    "DB_WW".WW_T_Auftrag_4; // AUFTRAG4 HOLEN I ->Z-HUB AUSGEFAHREN
      UN    "DB_WW".Schritt_T[7]; // SCHRITT7 SONDERSCHRITT
      UN    "I_WM_Taste_rechts"; // Rechtslauf WZ-Magazin
      UN    "I_WM_Taste_links"; // Linkslauf WZ-Magazin
      U(    ;
      O     "DB_WZV".Mag1_inPos_LST;
      O     "DB_ACHSE7".E_IndexAxisPos; // TEILUNGSACHSE WZ-MAG 1 IN POSITION
      O     "DB_WW".M1_LS_entsichern; // Freigabe Werkzeug entsichern Beladestation 1
      )     ;
      =     #FRG_WZ_MAN_RELEASE;

//      U     #FRG_WZ_MAN_RELEASE
//      UN    "I_WM_Energiefreigabe"      // Wz-Magazintür geschlossen
//      UN    "O_Bremse_oeffnen_Ax_7"     //"O_Bremse_oeffnen_Ax_7"// Bremse lüften WZ-Magazin 1
//      U     "I_WM_WZ_MAN_RELEASE"       // Fussschalter Werkzeughalter
//      O
//      U     "O_WM_WZ_ZYL_RELEASE"       // WZ-Halter öffnen (Beladestation) Magazin 1
//      U     "I_WM_WZ_MAN_RELEASE"       // Fussschalter Werkzeughalter
//      =     "O_WM_WZ_ZYL_RELEASE"       // WZ-Halter öffnen (Beladestation) Magazin 1

NETWORK
TITLE =WM_MagTasche: Werkzeug wurde an BELADESTATION entsichert
// BEFEHL DIE WZ-ZANGE OEFFNEN AM DER BELADESTATION MIT DEM
// FUSSSCHALTER
      U     "O_WM_WZ_ZYL_RELEASE"; // WZ-Halter öffnen (Beladestation) Magazin 1
      S     "DB_WW".M1_LS_entsichern; // Freigabe Werkzeug entsichern Beladestation 1

      U     #WZM_Fahrbefehl;
      R     "DB_WW".M1_LS_entsichern; // Freigabe Werkzeug entsichern Beladestation 1
      NOP   0;

NETWORK
TITLE ========== Werkzeug entspannen im Ablauf ===========



NETWORK
TITLE =WZ-Spanner: Einzelbewegung Freigabe Werkzeug entspannen

      O     #EB_Hand_WW;
      O     #Frg_Service;
      =     #EB_Frg_entspannen;
NETWORK
TITLE =WZ-Spanner: Einzelbewegung Werkzeug entspannen

      U     #EB_Frg_entspannen;
      U     "DB_EINRICHTFUNKTION".Bewegung_5_Minus;
      =     #EB_entspannen;

NETWORK
TITLE =WZ-Spanner: Einzelbewegung Freigabe Werkzeug spannen

      O     #EB_Hand_WW;
      O     #Frg_Service;
      =     #EB_Frg_spannen;

NETWORK
TITLE =WZ-Spanner: Einzelbewegung Werkzeug spannen

      U     #EB_Frg_spannen;
      U     "DB_EINRICHTFUNKTION".Bewegung_5_Plus;
      =     #EB_spannen;

NETWORK
TITLE =WZ-Spanner: Einzelbewegung Ansteuerung Anzeige
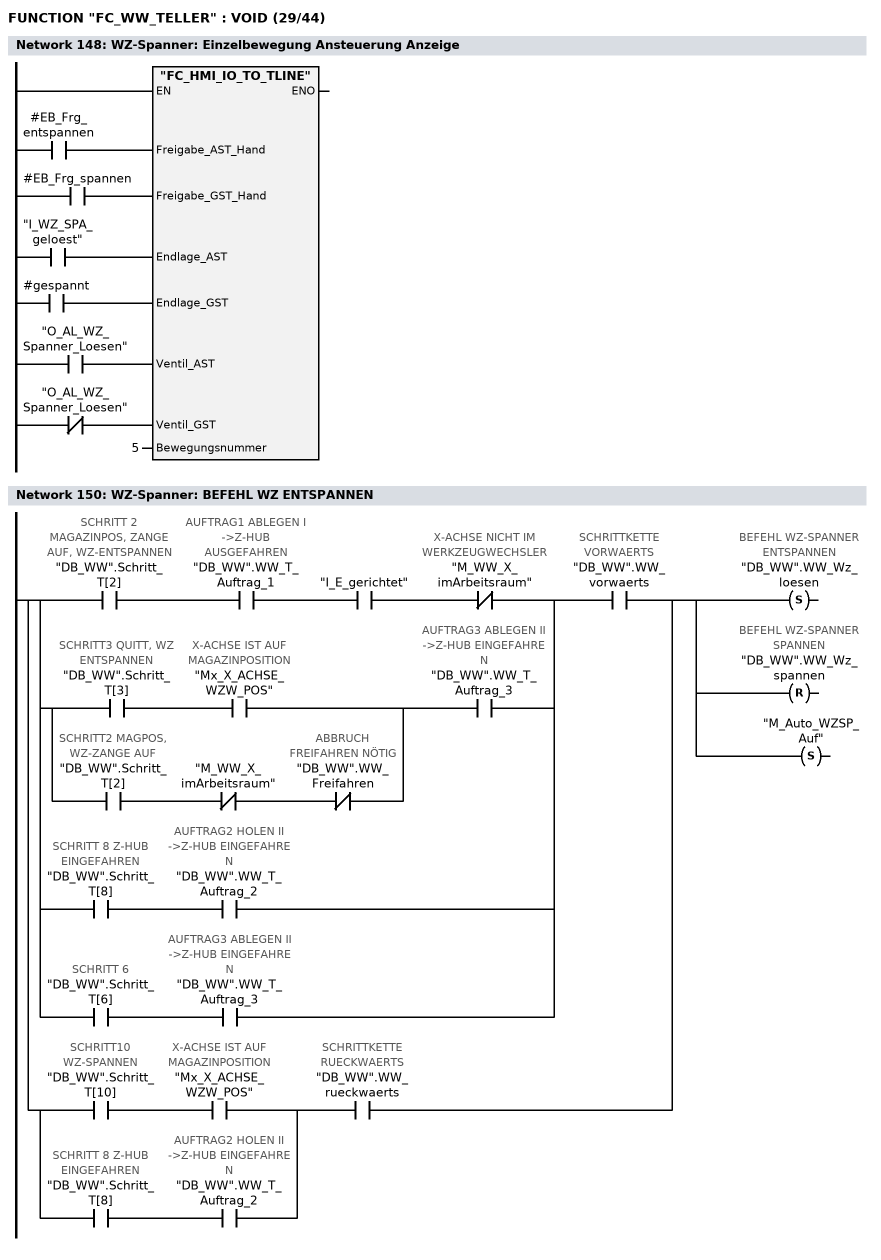

      U     #EB_Frg_entspannen;
      =     L     24.0;
      BLD   103;
      U     #EB_Frg_spannen;
      =     L     24.1;
      BLD   103;
      U     "I_WZ_SPA_geloest";
      =     L     24.2;
      BLD   103;
      U     #gespannt;
      =     L     24.3;
      BLD   103;
      U     "O_AL_WZ_Spanner_Loesen";
      =     L     24.4;
      BLD   103;
      UN    "O_AL_WZ_Spanner_Loesen";
      =     L     24.5;
      BLD   103;
      CALL "FC_HMI_IO_TO_TLINE" (
           Freigabe_AST_Hand        := L     24.0,
           Freigabe_GST_Hand        := L     24.1,
           Endlage_AST              := L     24.2,
           Endlage_GST              := L     24.3,
           Ventil_AST               := L     24.4,
           Ventil_GST               := L     24.5,
           Bewegungsnummer          := 5);
      NOP   0;
NETWORK
TITLE =WZ-Spanner: Einzelbewegung Ansteuerung Anzeige
//    U     #EB_Frg_entspannen
//      =     L24.0
//      BLD   103
//      U     #EB_Frg_spannen
//      =     #tx_Y_WP_frg
//      BLD   103
//      U     "I_WZ_SPA_geloest"
//      =     L24.2
//      BLD   103
//      U     #gespannt
//      =     L     24.3
//      BLD   103
//      U     "O_AL_WZ_Spanner_Loesen"
//      =     L     24.4
//      BLD   103
//      UN    "O_AL_WZ_Spanner_Loesen"
//      =     L     24.5
//      BLD   103
//      CALL  "FC_HMI_IO_TO_TLINE"
//       Freigabe_AST_Hand:=L24.0
//       Freigabe_GST_Hand:=#tx_Y_WP_frg
//       Endlage_AST      :=L24.2
//       Endlage_GST      :=L24.3
//       Ventil_AST       :=L24.4
//       Ventil_GST       :=L24.5
//       Bewegungsnummer  :=15
//      NOP   0
//


NETWORK
TITLE =WZ-Spanner: BEFEHL WZ ENTSPANNEN

      U(    ;
      U     "DB_WW".Schritt_T[2]; // SCHRITT 2 MAGAZINPOS, ZANGE AUF, WZ-ENTSPANNEN
      U     "DB_WW".WW_T_Auftrag_1; // AUFTRAG1 ABLEGEN I ->Z-HUB AUSGEFAHREN
      U     "I_E_gerichtet";
      UN    "M_WW_X_imArbeitsraum"; // X-ACHSE NICHT IM WERKZEUGWECHSLER
      O     ;
      U(    ;
      U     "DB_WW".Schritt_T[3]; // SCHRITT3 QUITT, WZ ENTSPANNEN
      U     "Mx_X_ACHSE_WZW_POS"; // X-ACHSE IST AUF MAGAZINPOSITION
      O     ;
      U     "DB_WW".Schritt_T[2]; // SCHRITT2 MAGPOS, WZ-ZANGE AUF
      UN    "M_WW_X_imArbeitsraum";
      UN    "DB_WW".WW_Freifahren; // ABBRUCH FREIFAHREN NÖTIG
      )     ;
      U     "DB_WW".WW_T_Auftrag_3; // AUFTRAG3 ABLEGEN II ->Z-HUB EINGEFAHREN
      O     ;
      U     "DB_WW".Schritt_T[8]; // SCHRITT 8 Z-HUB EINGEFAHREN
      U     "DB_WW".WW_T_Auftrag_2; // AUFTRAG2 HOLEN II ->Z-HUB EINGEFAHREN
      O     ;
      U     "DB_WW".Schritt_T[6]; // SCHRITT 6
      U     "DB_WW".WW_T_Auftrag_3; // AUFTRAG3 ABLEGEN II ->Z-HUB EINGEFAHREN
      )     ;
      U     "DB_WW".WW_vorwaerts; // SCHRITTKETTE VORWAERTS
      O     ;
      U(    ;
      U     "DB_WW".Schritt_T[10]; // SCHRITT10 WZ-SPANNEN
      U     "Mx_X_ACHSE_WZW_POS"; // X-ACHSE IST AUF MAGAZINPOSITION
      O     ;
      U     "DB_WW".Schritt_T[8]; // SCHRITT 8 Z-HUB EINGEFAHREN
      U     "DB_WW".WW_T_Auftrag_2; // AUFTRAG2 HOLEN II ->Z-HUB EINGEFAHREN
      )     ;
      U     "DB_WW".WW_rueckwaerts; // SCHRITTKETTE RUECKWAERTS
      S     "DB_WW".WW_Wz_loesen; // BEFEHL WZ-SPANNER ENTSPANNEN
      R     "DB_WW".WW_Wz_spannen; // BEFEHL WZ-SPANNER SPANNEN
      S     "M_Auto_WZSP_Auf";

NETWORK
TITLE =WZ-Spanner: BEFEHL WZ SPANNEN
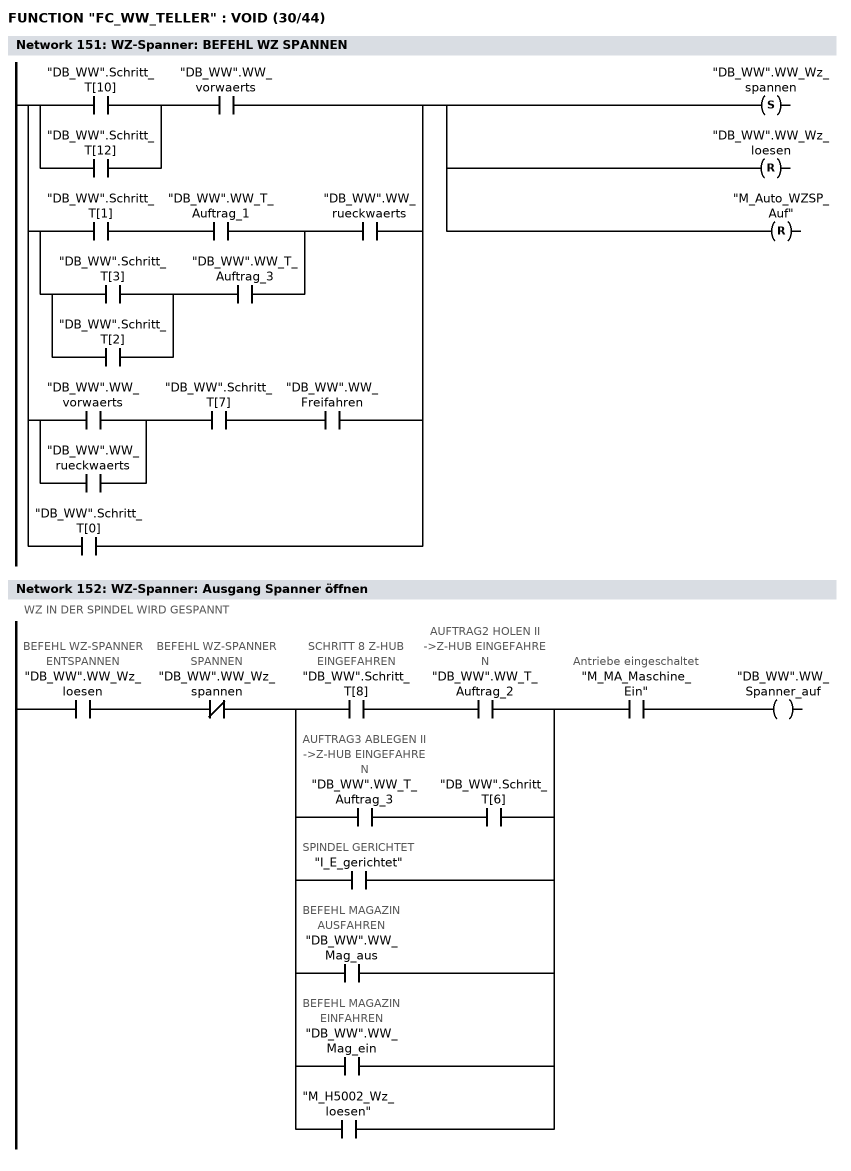

      U(    ;
      O     "DB_WW".Schritt_T[10];
      O     "DB_WW".Schritt_T[12];
      )     ;
      U     "DB_WW".WW_vorwaerts;
      O     ;
      U(    ;
      U     "DB_WW".Schritt_T[1];
      U     "DB_WW".WW_T_Auftrag_1;
      O     ;
      U(    ;
      O     "DB_WW".Schritt_T[3];
      O     "DB_WW".Schritt_T[2];
      )     ;
      U     "DB_WW".WW_T_Auftrag_3;
      )     ;
      U     "DB_WW".WW_rueckwaerts;
      O     ;
      U(    ;
      O     "DB_WW".WW_vorwaerts;
      O     "DB_WW".WW_rueckwaerts;
      )     ;
      U     "DB_WW".Schritt_T[7];
      U     "DB_WW".WW_Freifahren;
      O     "DB_WW".Schritt_T[0];
      S     "DB_WW".WW_Wz_spannen;
      R     "DB_WW".WW_Wz_loesen;
      R     "M_Auto_WZSP_Auf";

NETWORK
TITLE =WZ-Spanner: Ausgang Spanner öffnen
// WZ IN DER SPINDEL WIRD GESPANNT
      U     "DB_WW".WW_Wz_loesen; // BEFEHL WZ-SPANNER ENTSPANNEN
      UN    "DB_WW".WW_Wz_spannen; // BEFEHL WZ-SPANNER SPANNEN
      U(    ;
      U     "DB_WW".Schritt_T[8]; // SCHRITT 8 Z-HUB EINGEFAHREN
      U     "DB_WW".WW_T_Auftrag_2; // AUFTRAG2 HOLEN II ->Z-HUB EINGEFAHREN
      O     ;
      U     "DB_WW".WW_T_Auftrag_3; // AUFTRAG3 ABLEGEN II ->Z-HUB EINGEFAHREN
      U     "DB_WW".Schritt_T[6];
      O     "I_E_gerichtet"; // SPINDEL GERICHTET
      O     "DB_WW".WW_Mag_aus; // BEFEHL MAGAZIN AUSFAHREN
      O     "DB_WW".WW_Mag_ein; // BEFEHL MAGAZIN EINFAHREN
      O     "M_H5002_Wz_loesen";
      )     ;
      U     "M_MA_Maschine_Ein"; // Antriebe eingeschaltet
      =     "DB_WW".WW_Spanner_auf;
NETWORK
TITLE =Ausgang SPINDELKONUS AUSBLASEN
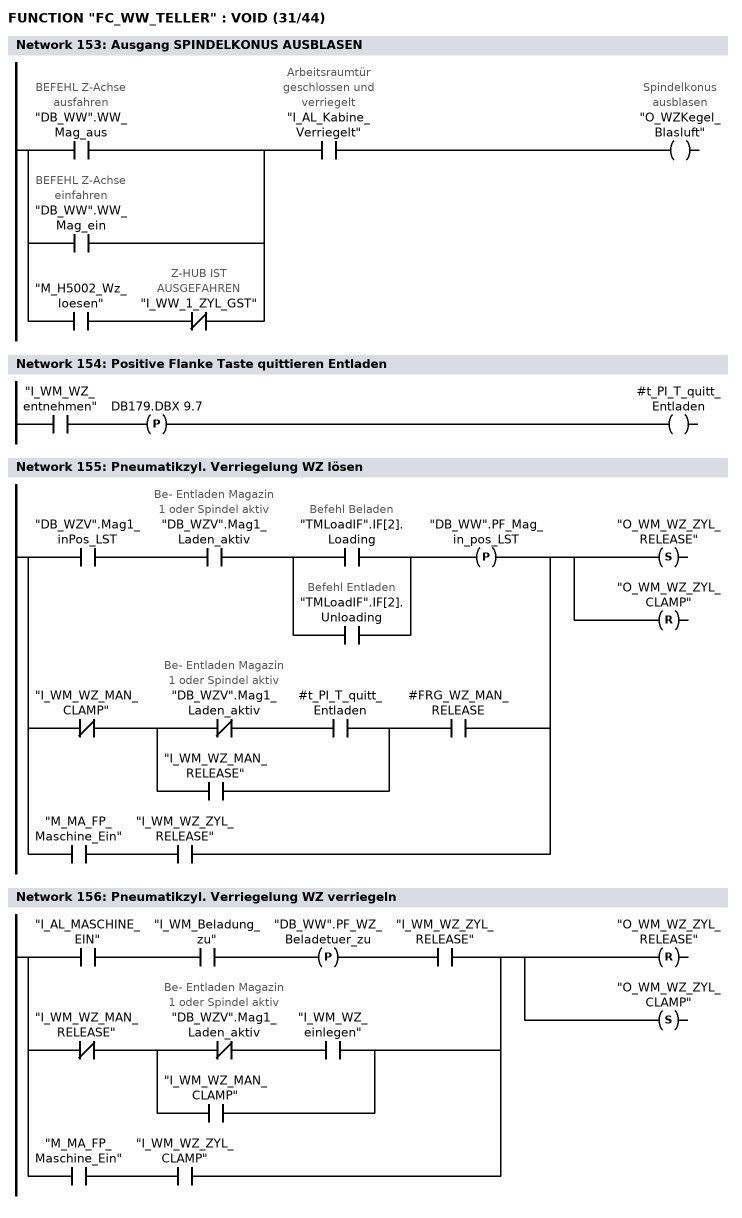

      U(    ;
      O     "DB_WW".WW_Mag_aus; // BEFEHL Z-Achse ausfahren
      O     "DB_WW".WW_Mag_ein; // BEFEHL Z-Achse einfahren
      O     ;
      U     "M_H5002_Wz_loesen";
      UN    "I_WW_1_ZYL_GST"; // Z-HUB IST AUSGEFAHREN
      )     ;
      U     "I_AL_Kabine_Verriegelt"; // Arbeitsraumtür geschlossen und verriegelt
      =     "O_WZKegel_Blasluft"; // Spindelkonus ausblasen

NETWORK
TITLE =Positive Flanke Taste quittieren Entladen

      U     "I_WM_WZ_entnehmen";
      FP    DB179.DBX    9.7;
      =     #t_PI_T_quitt_Entladen;
NETWORK
TITLE =Pneumatikzyl. Verriegelung WZ lösen

      U     "DB_WZV".Mag1_inPos_LST;
      U     "DB_WZV".Mag1_Laden_aktiv; // Be- Entladen Magazin 1 oder Spindel aktiv
      U(    ;
      O     "TMLoadIF".IF[2].Loading; // Befehl Beladen
      O     "TMLoadIF".IF[2].Unloading; // Befehl Entladen
      )     ;
      FP    "DB_WW".PF_Mag_in_pos_LST;
      O     ;
      UN    "I_WM_WZ_MAN_CLAMP";
      U(    ;
      UN    "DB_WZV".Mag1_Laden_aktiv; // Be- Entladen Magazin 1 oder Spindel aktiv
      U     #t_PI_T_quitt_Entladen;
      O     "I_WM_WZ_MAN_RELEASE";
      )     ;
      U     #FRG_WZ_MAN_RELEASE;
      O     ;

      U     "M_MA_FP_Maschine_Ein";
      U     "I_WM_WZ_ZYL_RELEASE";
      S     "O_WM_WZ_ZYL_RELEASE";
      R     "O_WM_WZ_ZYL_CLAMP";
NETWORK
TITLE =Pneumatikzyl. Verriegelung WZ verriegeln

      U     "I_AL_MASCHINE_EIN";
      U     "I_WM_Beladung_zu";
      FP    "DB_WW".PF_WZ_Beladetuer_zu;
      U     "I_WM_WZ_ZYL_RELEASE";
      O     ;

      UN    "I_WM_WZ_MAN_RELEASE";
      U(    ;
      UN    "DB_WZV".Mag1_Laden_aktiv; // Be- Entladen Magazin 1 oder Spindel aktiv
      U     "I_WM_WZ_einlegen";
      O     "I_WM_WZ_MAN_CLAMP";
      )     ;
      O     ;
      U     "M_MA_FP_Maschine_Ein";
      U     "I_WM_WZ_ZYL_CLAMP";
      R     "O_WM_WZ_ZYL_RELEASE";
      S     "O_WM_WZ_ZYL_CLAMP";
NETWORK
TITLE ========== Vorschubsperren ===============



NETWORK
TITLE =VSP, alle Achsen
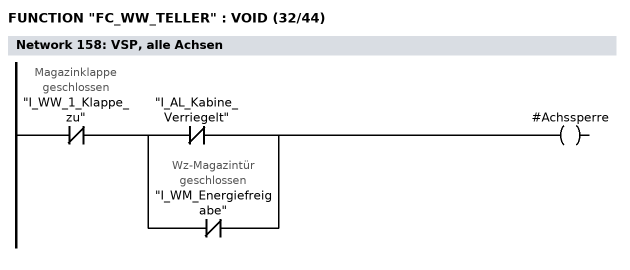

      UN    "I_WW_1_Klappe_zu"; // Magazinklappe geschlossen
      U(    ;
      ON    "I_AL_Kabine_Verriegelt";
      ON    "I_WM_Energiefreigabe"; // Wz-Magazintür geschlossen
      )     ;
      =     #Achssperre;

NETWORK
TITLE =VSP-X, Werkzeugwechsler
//Die X-Achse soll bei Überschreiten der Warteposition gesperrt werden:
//1. Wenn kein Verfahrschritt (1,2,7,11,12) und kein Werkzeugvermessen ansteht,
//   ausser der Wechsler ist noch nicht initialisiert (kein Schrittmerker) oder
//
//   ist in Grundstellung oder es steht Werkzeugvermessen an. Dann darf die
//   Freigabe aber auch nur im JOG und mit Fahrbefehl X- gegeben werden.
//2. Wenn im Schritt 7 Automatik ansteht oder im Freifahrmodus Fahrbefehl X-
//   ansteht.
//3. Wenn im Schritt 1,2,11 oder 12 im Freifahrmodus Fahrbefehl X- ansteht.
//4. Wenn im Schritt 1 oder 2 die Spindel nicht gerichtet ist. (nur AUTO)
//5. Wenn die Magazinklappe nicht geöffnet ist.(nur bei elektrischer Klappe)
//6. Wenn im Verfahrschritt keine Freigabe Ausgänge ansteht
//7. Wenn im Schritt 2 oder 11 die Werkzeugtasche nicht verriegelt ist.
//
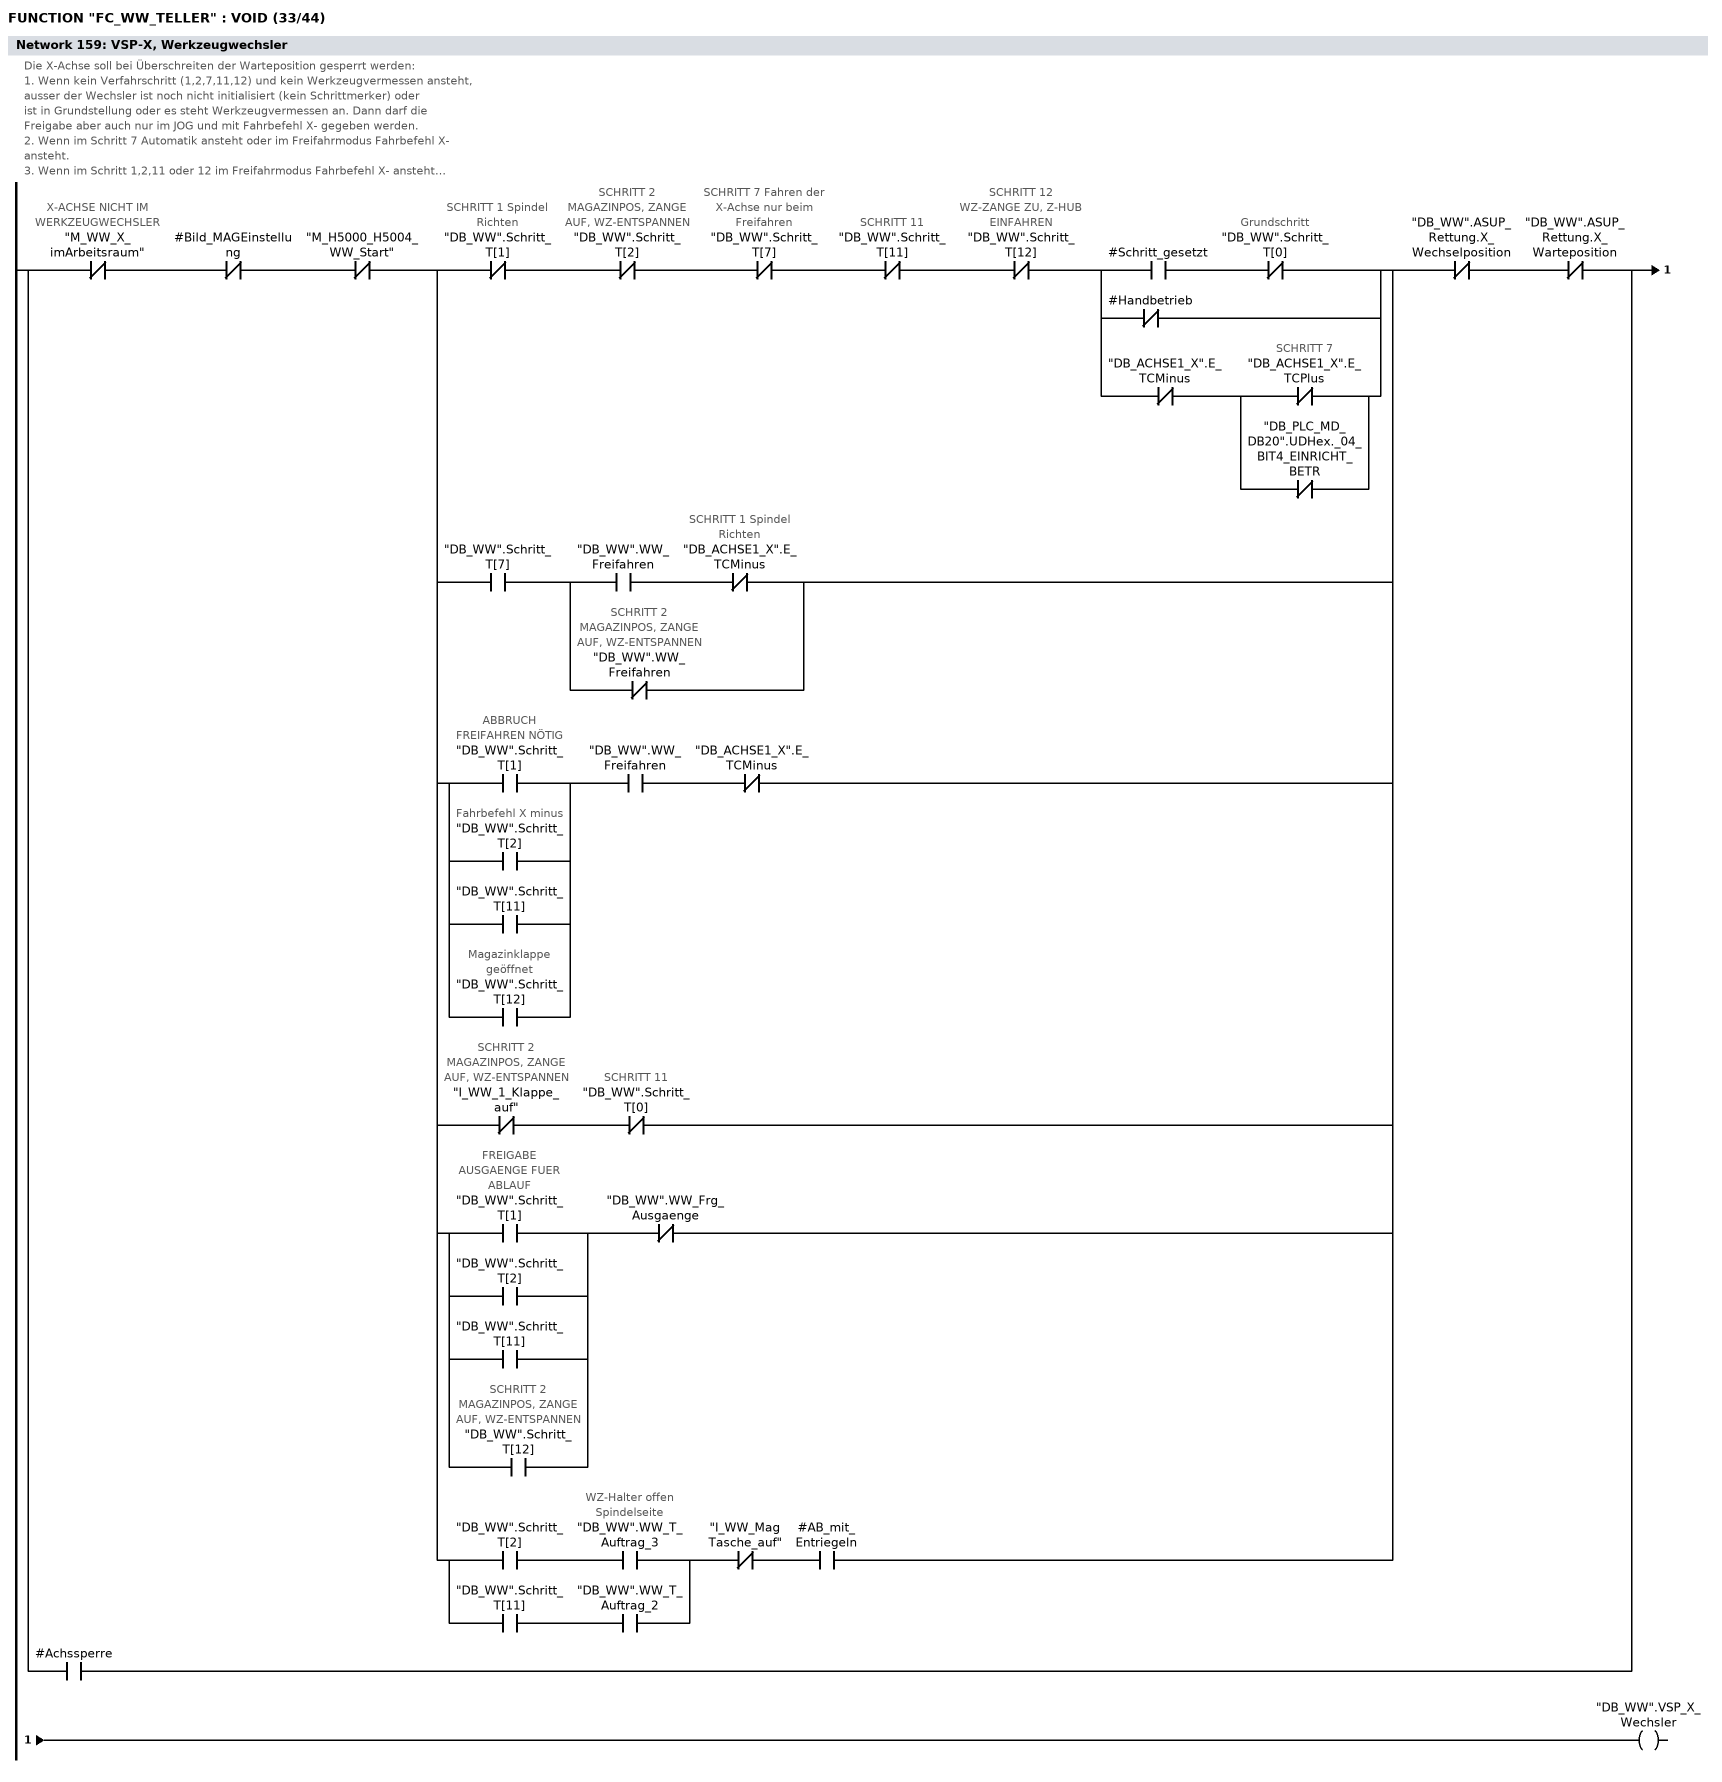
      UN    "M_WW_X_imArbeitsraum"; // X-ACHSE NICHT IM WERKZEUGWECHSLER
      UN    #Bild_MAGEinstellung;
      UN    "M_H5000_H5004_WW_Start";
      U(    ;

      UN    "DB_WW".Schritt_T[1]; // SCHRITT 1 Spindel Richten
      UN    "DB_WW".Schritt_T[2]; // SCHRITT 2 MAGAZINPOS, ZANGE AUF, WZ-ENTSPANNEN
      UN    "DB_WW".Schritt_T[7]; // SCHRITT 7 Fahren der X-Achse nur beim Freifahren
      UN    "DB_WW".Schritt_T[11]; // SCHRITT 11
      UN    "DB_WW".Schritt_T[12]; // SCHRITT 12 WZ-ZANGE ZU, Z-HUB EINFAHREN
      U(    ;
      U     #Schritt_gesetzt;
      UN    "DB_WW".Schritt_T[0]; // Grundschritt
      ON    #Handbetrieb;
      O     ; // Fahrbefehl X minus
      UN    "DB_ACHSE1_X".E_TCMinus;

      U(    ;
      ON    "DB_ACHSE1_X".E_TCPlus; // SCHRITT 7
      ON    "DB_PLC_MD_DB20".UDHex._04_BIT4_EINRICHT_BETR;
      )     ; // ABBRUCH FREIFAHREN NÖTIG
      )     ; // Fahrbefehl X minus
      O     ; // ABBRUCH FREIFAHREN NÖTIG
      U     "DB_WW".Schritt_T[7];

      U(    ;
      U     "DB_WW".WW_Freifahren;
      UN    "DB_ACHSE1_X".E_TCMinus; // SCHRITT 1 Spindel Richten
      ON    "DB_WW".WW_Freifahren; // SCHRITT 2 MAGAZINPOS, ZANGE AUF, WZ-ENTSPANNEN
      )     ; // SCHRITT 11
      O     ; // SCHRITT 12 WZ-ZANGE ZU, Z-HUB EINFAHREN
      U(    ;
      O     "DB_WW".Schritt_T[1]; // ABBRUCH FREIFAHREN NÖTIG
      O     "DB_WW".Schritt_T[2]; // Fahrbefehl X minus

      O     "DB_WW".Schritt_T[11];
      O     "DB_WW".Schritt_T[12]; // Magazinklappe geöffnet
      )     ; // Grundschritt

      U     "DB_WW".WW_Freifahren;
      UN    "DB_ACHSE1_X".E_TCMinus;
      O     ; // SCHRITT 1 Spindel Richten
      UN    "I_WW_1_Klappe_auf"; // SCHRITT 2 MAGAZINPOS, ZANGE AUF, WZ-ENTSPANNEN
      UN    "DB_WW".Schritt_T[0]; // SCHRITT 11
      O     ; // SCHRITT 12 WZ-ZANGE ZU, Z-HUB EINFAHREN
      U(    ;
      O     "DB_WW".Schritt_T[1]; // FREIGABE AUSGAENGE FUER ABLAUF

      O     "DB_WW".Schritt_T[2];
      O     "DB_WW".Schritt_T[11];
      O     "DB_WW".Schritt_T[12]; // SCHRITT 2 MAGAZINPOS, ZANGE AUF, WZ-ENTSPANNEN
      )     ; // AUFTRAG3 ABLEGEN II ->Z-HUB EINGEFAHREN
      UN    "DB_WW".WW_Frg_Ausgaenge;
      O     ; // SCHRITT11 WZ-ZANGE AUF, X-ACHSE WARTPOS
      U(    ; // AUFTRAG2 HOLEN II ->Z-HUB EINGEFAHREN
      U     "DB_WW".Schritt_T[2];
      U     "DB_WW".WW_T_Auftrag_3; // WZ-Halter offen Spindelseite
      O     ;

      U     "DB_WW".Schritt_T[11];
      U     "DB_WW".WW_T_Auftrag_2;
      )     ;
      UN    "I_WW_MagTasche_auf";
      U     #AB_mit_Entriegeln;

      )     ;
      UN    "DB_WW".ASUP_Rettung.X_Wechselposition;
      UN    "DB_WW".ASUP_Rettung.X_Warteposition;
      O     #Achssperre;
      =     "DB_WW".VSP_X_Wechsler;
NETWORK
TITLE =_701303 Vorschubsperre X Werkzeugwechsler
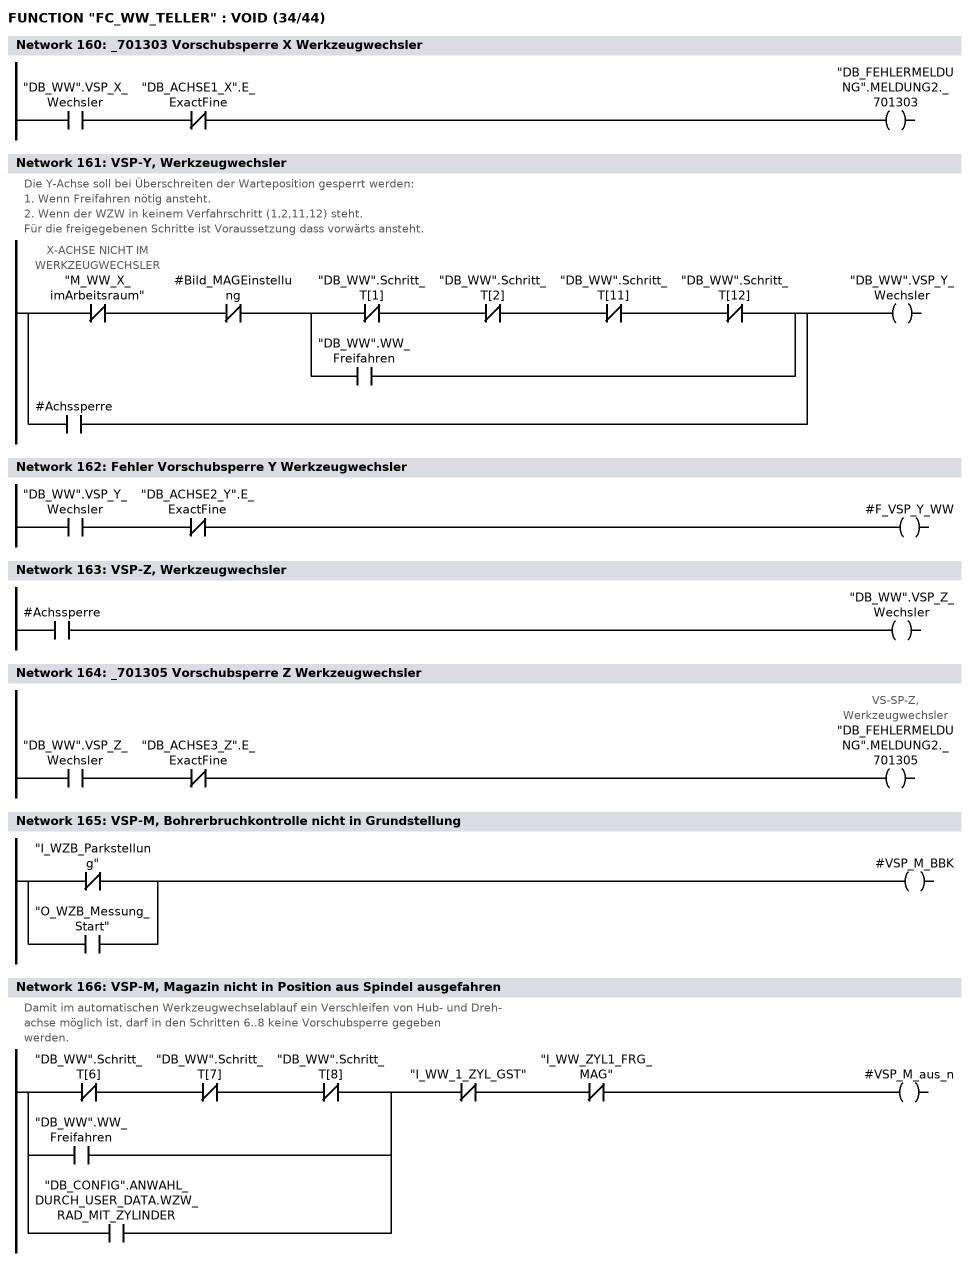

      U     "DB_WW".VSP_X_Wechsler;
      UN    "DB_ACHSE1_X".E_ExactFine;
      =     "DB_FEHLERMELDUNG".MELDUNG2._701303;

NETWORK
TITLE =VSP-Y, Werkzeugwechsler
// Die Y-Achse soll bei Überschreiten der Warteposition gesperrt werden:
// 1. Wenn Freifahren nötig ansteht.
// 2. Wenn der WZW in keinem Verfahrschritt (1,2,11,12) steht.
//    Für die freigegebenen Schritte ist Voraussetzung dass vorwärts ansteht.
      UN    "M_WW_X_imArbeitsraum"; // X-ACHSE NICHT IM WERKZEUGWECHSLER
      UN    #Bild_MAGEinstellung;
      U(    ;
      UN    "DB_WW".Schritt_T[1];
      UN    "DB_WW".Schritt_T[2];
      UN    "DB_WW".Schritt_T[11];
      UN    "DB_WW".Schritt_T[12];
//      ON    "DB_WW".WW_vorwaerts
      O     "DB_WW".WW_Freifahren;
      )     ;
      O     #Achssperre;
      =     "DB_WW".VSP_Y_Wechsler;

NETWORK
TITLE =Fehler Vorschubsperre Y Werkzeugwechsler

      U     "DB_WW".VSP_Y_Wechsler;
      UN    "DB_ACHSE2_Y".E_ExactFine;
      =     #F_VSP_Y_WW;

NETWORK
TITLE =VSP-Z, Werkzeugwechsler

      U     #Achssperre;
      =     "DB_WW".VSP_Z_Wechsler;

NETWORK
TITLE =_701305 Vorschubsperre Z Werkzeugwechsler

      U     "DB_WW".VSP_Z_Wechsler;
      UN    "DB_ACHSE3_Z".E_ExactFine;
      =     "DB_FEHLERMELDUNG".MELDUNG2._701305; // VS-SP-Z, Werkzeugwechsler

NETWORK
TITLE =VSP-M, Bohrerbruchkontrolle nicht in Grundstellung

      ON    "I_WZB_Parkstellung";
      O     "O_WZB_Messung_Start";
      =     #VSP_M_BBK;
NETWORK
TITLE =VSP-M, Magazin nicht in Position aus Spindel ausgefahren
//Damit im automatischen Werkzeugwechselablauf ein Verschleifen von Hub- und Dreh-
//achse möglich ist, darf in den Schritten 6..8 keine Vorschubsperre gegeben
//werden.
      U(    ;
      UN    "DB_WW".Schritt_T[6];
      UN    "DB_WW".Schritt_T[7];
      UN    "DB_WW".Schritt_T[8];
      O     "DB_WW".WW_Freifahren;
      O     "DB_CONFIG".ANWAHL_DURCH_USER_DATA.WZW_RAD_MIT_ZYLINDER;
      )     ;
      UN    "I_WW_1_ZYL_GST";
      UN    "I_WW_ZYL1_FRG_MAG";
      =     #VSP_M_aus_n;
NETWORK
TITLE =VSP-M, Werkzeugwechsler
// FREIGABE ZUM DREHEN DES MAGAZIN. BEI FEHLEN VON MERKER M76.3 MUSS
// ACHSE DES MAGAZINS SOFORT STEHEN BLEIBEN.
//   ON    "I_WM_WZ_ZYL_CLAMP"         // WZ-Halter geschlossen
//    ON    #HalterSp_zu
//   U     "DB_ACHSE7".E_IndexAxisPos  // "DB_ACHSE7".E_ExactFine
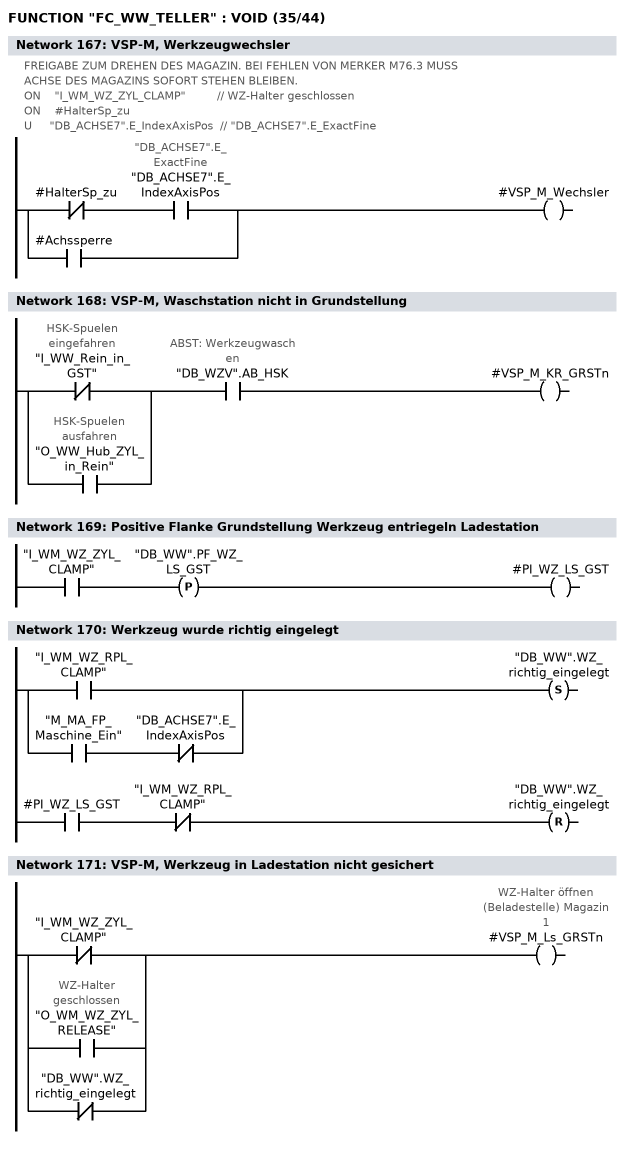
      UN    #HalterSp_zu;
      U     "DB_ACHSE7".E_IndexAxisPos; // "DB_ACHSE7".E_ExactFine
      O     #Achssperre;
      =     #VSP_M_Wechsler;

NETWORK
TITLE =VSP-M, Waschstation nicht in Grundstellung

      U(    ;
      ON    "I_WW_Rein_in_GST"; // HSK-Spuelen eingefahren
      O     "O_WW_Hub_ZYL_in_Rein"; // HSK-Spuelen ausfahren
      )     ;
      U     "DB_WZV".AB_HSK; // ABST: Werkzeugwaschen
      =     #VSP_M_KR_GRSTn;

NETWORK
TITLE =Positive Flanke Grundstellung Werkzeug entriegeln Ladestation

      U     "I_WM_WZ_ZYL_CLAMP";
      FP    "DB_WW".PF_WZ_LS_GST;
      =     #PI_WZ_LS_GST;

NETWORK
TITLE =Werkzeug wurde richtig eingelegt

      U(    ;
      O     "I_WM_WZ_RPL_CLAMP";
      O     ;
      U     "M_MA_FP_Maschine_Ein";
      UN    "DB_ACHSE7".E_IndexAxisPos;
      )     ;
      S     "DB_WW".WZ_richtig_eingelegt;
      U     #PI_WZ_LS_GST;
      UN    "I_WM_WZ_RPL_CLAMP";
      R     "DB_WW".WZ_richtig_eingelegt;
      NOP   0;
NETWORK
TITLE =VSP-M, Werkzeug in Ladestation nicht gesichert
//
      ON    "I_WM_WZ_ZYL_CLAMP";
      O     "O_WM_WZ_ZYL_RELEASE"; // WZ-Halter geschlossen
      ON    "DB_WW".WZ_richtig_eingelegt;
      =     #VSP_M_Ls_GRSTn; // WZ-Halter öffnen (Beladestelle) Magazin 1
NETWORK
TITLE =VSP-M, Werkzeugwechsler
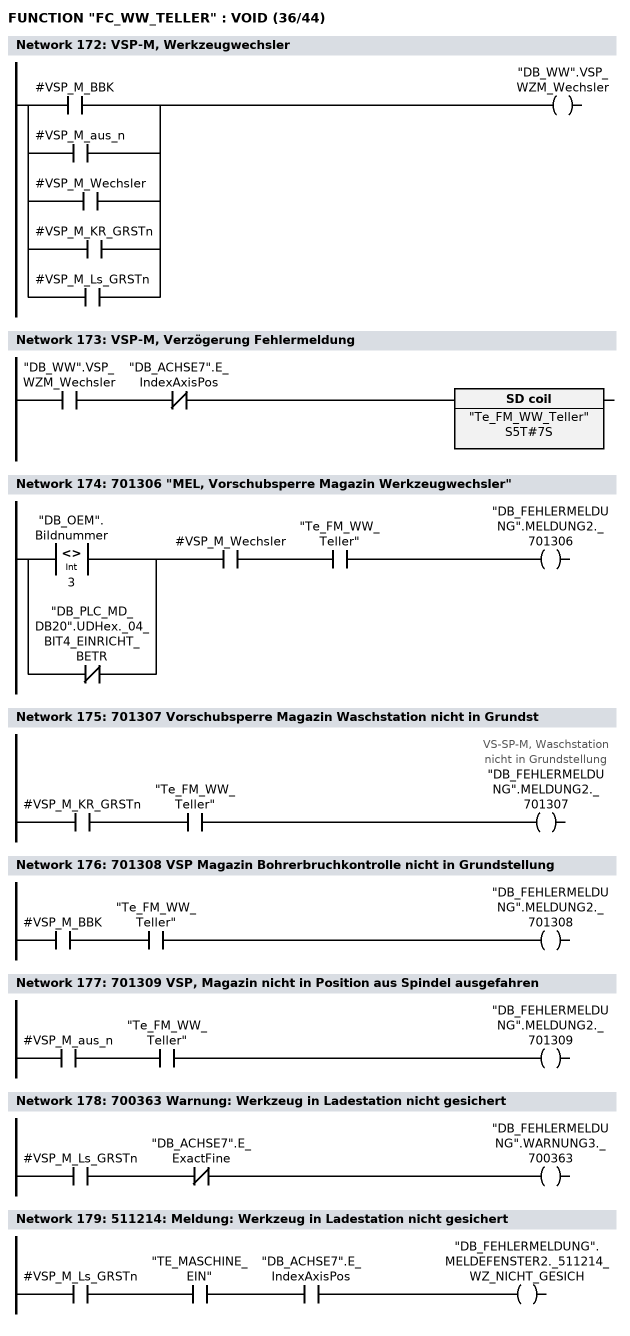

      O     #VSP_M_BBK;
      O     #VSP_M_aus_n;
      O     #VSP_M_Wechsler;
      O     #VSP_M_KR_GRSTn;
      O     #VSP_M_Ls_GRSTn;
      =     "DB_WW".VSP_WZM_Wechsler;

NETWORK
TITLE =VSP-M, Verzögerung Fehlermeldung

      U     "DB_WW".VSP_WZM_Wechsler;
      UN    "DB_ACHSE7".E_IndexAxisPos;
      L     S5T#7S;
      SE    "Te_FM_WW_Teller";

NETWORK
TITLE =701306 "MEL, Vorschubsperre Magazin Werkzeugwechsler"

      U(    ;
      O(    ;
      L     "DB_OEM".Bildnummer;
      L     3;
      <>I   ;
      )     ;
      ON    "DB_PLC_MD_DB20".UDHex._04_BIT4_EINRICHT_BETR;
      )     ;
      U     #VSP_M_Wechsler;
      U     "Te_FM_WW_Teller";
      =     "DB_FEHLERMELDUNG".MELDUNG2._701306;
NETWORK
TITLE =701307 Vorschubsperre Magazin Waschstation nicht in Grundst

      U     #VSP_M_KR_GRSTn;
      U     "Te_FM_WW_Teller";
      =     "DB_FEHLERMELDUNG".MELDUNG2._701307; // VS-SP-M, Waschstation nicht in Grundstellung

NETWORK
TITLE =701308 VSP Magazin Bohrerbruchkontrolle nicht in Grundstellung

      U     #VSP_M_BBK;
      U     "Te_FM_WW_Teller";
      =     "DB_FEHLERMELDUNG".MELDUNG2._701308;

NETWORK
TITLE =701309 VSP, Magazin nicht in Position aus Spindel ausgefahren

      U     #VSP_M_aus_n;
      U     "Te_FM_WW_Teller";
      =     "DB_FEHLERMELDUNG".MELDUNG2._701309;

NETWORK
TITLE =700363 Warnung: Werkzeug in Ladestation nicht gesichert

      U     #VSP_M_Ls_GRSTn;
      UN    "DB_ACHSE7".E_ExactFine;
      =     "DB_FEHLERMELDUNG".WARNUNG3._700363;

NETWORK
TITLE =511214: Meldung: Werkzeug in Ladestation nicht gesichert

      U     #VSP_M_Ls_GRSTn;
      U     "TE_MASCHINE_EIN";
      U     "DB_ACHSE7".E_IndexAxisPos;
      =     "DB_FEHLERMELDUNG".MELDEFENSTER2._511214_WZ_NICHT_GESICH;
NETWORK
TITLE =_700434 VS-H, ENDSCHALTERSTOERUNG Werkzeugwechsel
// FEHLERAUSWERTUNG DER EINGAENGE DES WZ-WECHSLERS
// 1.TEIL GEGENSEITIGE AUSWERTUNG -> VSP
// 2.TEIL WARTEN AUF RUECKMELDUNGEN -> NUR ANZEIGE
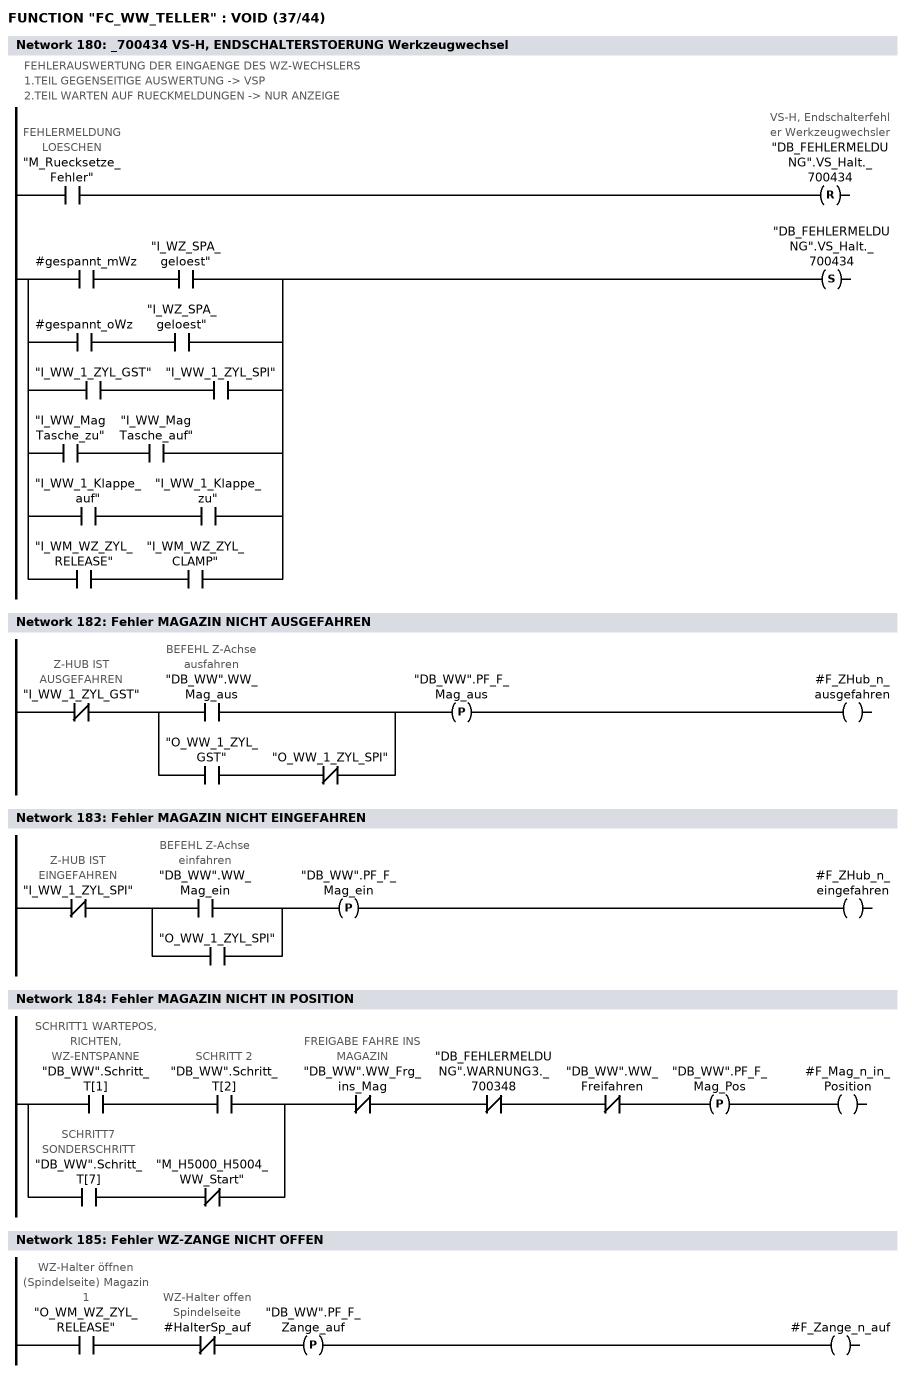
      U     "M_Ruecksetze_Fehler"; // FEHLERMELDUNG LOESCHEN
      R     "DB_FEHLERMELDUNG".VS_Halt._700434; // VS-H, Endschalterfehler Werkzeugwechsler

      U(    ;
      U     #gespannt_mWz;
      U     "I_WZ_SPA_geloest";
      O     ;
      U     #gespannt_oWz;
      U     "I_WZ_SPA_geloest";
      O     ;
      U     "I_WW_1_ZYL_GST";
      U     "I_WW_1_ZYL_SPI";
      O     ;
      U     "I_WW_MagTasche_zu";
      U     "I_WW_MagTasche_auf";
      O     ;
      U     "I_WW_1_Klappe_auf";
      U     "I_WW_1_Klappe_zu";
      O     ;

      U     "I_WM_WZ_ZYL_RELEASE";
      U     "I_WM_WZ_ZYL_CLAMP";
      )     ;
      S     "DB_FEHLERMELDUNG".VS_Halt._700434;
      NOP   0;
NETWORK
TITLE ============= Überwachung Endposition ==========



NETWORK
TITLE =Fehler MAGAZIN NICHT AUSGEFAHREN

      UN    "I_WW_1_ZYL_GST"; // Z-HUB IST AUSGEFAHREN
      U(    ;
      O     "DB_WW".WW_Mag_aus; // BEFEHL Z-Achse ausfahren
      O     ;
      U     "O_WW_1_ZYL_GST";
      UN    "O_WW_1_ZYL_SPI";
      )     ;

      FP    "DB_WW".PF_F_Mag_aus;
      =     #F_ZHub_n_ausgefahren;
NETWORK
TITLE =Fehler MAGAZIN NICHT EINGEFAHREN

      UN    "I_WW_1_ZYL_SPI"; // Z-HUB IST EINGEFAHREN
      U(    ;
      O     "DB_WW".WW_Mag_ein; // BEFEHL Z-Achse einfahren
      O     "O_WW_1_ZYL_SPI";
      )     ;
      FP    "DB_WW".PF_F_Mag_ein;
      =     #F_ZHub_n_eingefahren;

NETWORK
TITLE =Fehler MAGAZIN NICHT IN POSITION

      U(    ;
      U     "DB_WW".Schritt_T[1]; // SCHRITT1 WARTEPOS, RICHTEN, WZ-ENTSPANNE
      U     "DB_WW".Schritt_T[2]; // SCHRITT 2
      O     ;
      U     "DB_WW".Schritt_T[7]; // SCHRITT7 SONDERSCHRITT
      UN    "M_H5000_H5004_WW_Start";
      )     ;
      UN    "DB_WW".WW_Frg_ins_Mag; // FREIGABE FAHRE INS MAGAZIN
      UN    "DB_FEHLERMELDUNG".WARNUNG3._700348;
      UN    "DB_WW".WW_Freifahren;
      FP    "DB_WW".PF_F_Mag_Pos;
      =     #F_Mag_n_in_Position;

NETWORK
TITLE =Fehler WZ-ZANGE NICHT OFFEN

      U     "O_WM_WZ_ZYL_RELEASE"; // WZ-Halter öffnen (Spindelseite) Magazin 1
      UN    #HalterSp_auf; // WZ-Halter offen Spindelseite
      FP    "DB_WW".PF_F_Zange_auf;
      =     #F_Zange_n_auf;

NETWORK
TITLE =Fehler WZ-ZANGE NICHT GESCHLOSSEN
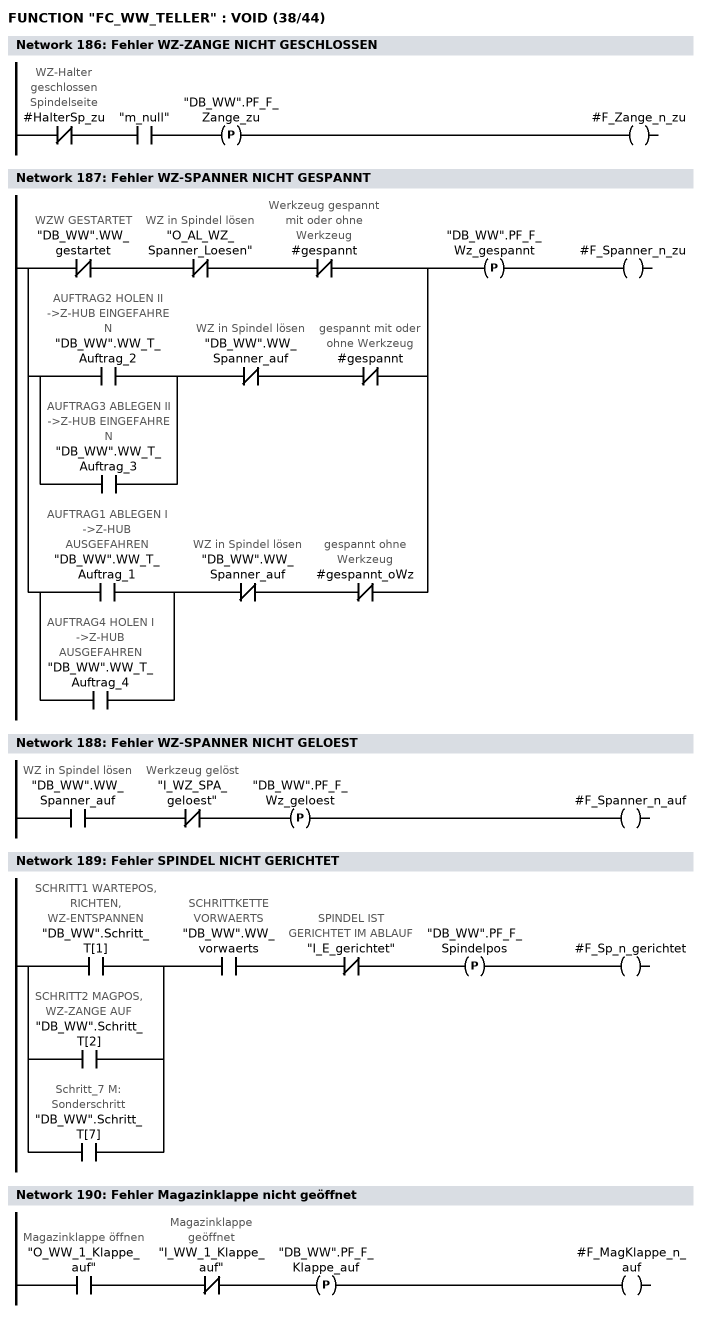

      UN    #HalterSp_zu; // WZ-Halter geschlossen Spindelseite
      U     "m_null";
      FP    "DB_WW".PF_F_Zange_zu;
      =     #F_Zange_n_zu;

NETWORK
TITLE =Fehler WZ-SPANNER NICHT GESPANNT

      UN    "DB_WW".WW_gestartet; // WZW GESTARTET
      UN    "O_AL_WZ_Spanner_Loesen"; // WZ in Spindel lösen
      UN    #gespannt; // Werkzeug gespannt mit oder ohne Werkzeug
      O     ;
      U(    ;
      O     "DB_WW".WW_T_Auftrag_2; // AUFTRAG2 HOLEN II ->Z-HUB EINGEFAHREN
      O     "DB_WW".WW_T_Auftrag_3; // AUFTRAG3 ABLEGEN II ->Z-HUB EINGEFAHREN
      )     ;
      UN    "DB_WW".WW_Spanner_auf; // WZ in Spindel lösen
      UN    #gespannt; // gespannt mit oder ohne Werkzeug
      O     ;
      U(    ;
      O     "DB_WW".WW_T_Auftrag_1; // AUFTRAG1 ABLEGEN I ->Z-HUB AUSGEFAHREN
      O     "DB_WW".WW_T_Auftrag_4; // AUFTRAG4 HOLEN I ->Z-HUB AUSGEFAHREN
      )     ;
      UN    "DB_WW".WW_Spanner_auf; // WZ in Spindel lösen
      UN    #gespannt_oWz; // gespannt ohne Werkzeug
      FP    "DB_WW".PF_F_Wz_gespannt;
      =     #F_Spanner_n_zu;

NETWORK
TITLE =Fehler WZ-SPANNER NICHT GELOEST

      U     "DB_WW".WW_Spanner_auf; // WZ in Spindel lösen
      UN    "I_WZ_SPA_geloest"; // Werkzeug gelöst
      FP    "DB_WW".PF_F_Wz_geloest;
      =     #F_Spanner_n_auf;

NETWORK
TITLE =Fehler SPINDEL NICHT GERICHTET

      U(    ;
      O     "DB_WW".Schritt_T[1]; // SCHRITT1 WARTEPOS, RICHTEN, WZ-ENTSPANNEN
      O     "DB_WW".Schritt_T[2]; // SCHRITT2 MAGPOS, WZ-ZANGE AUF
      O     "DB_WW".Schritt_T[7]; // Schritt_7 M: Sonderschritt
      )     ;
      U     "DB_WW".WW_vorwaerts; // SCHRITTKETTE VORWAERTS
      UN    "I_E_gerichtet"; // SPINDEL IST GERICHTET IM ABLAUF
      FP    "DB_WW".PF_F_Spindelpos;
      =     #F_Sp_n_gerichtet;

NETWORK
TITLE =Fehler Magazinklappe nicht geöffnet

      U     "O_WW_1_Klappe_auf"; // Magazinklappe öffnen
      UN    "I_WW_1_Klappe_auf"; // Magazinklappe geöffnet
      FP    "DB_WW".PF_F_Klappe_auf;
      =     #F_MagKlappe_n_auf;

NETWORK
TITLE =Fehler Magazinklappe nicht geschlossen
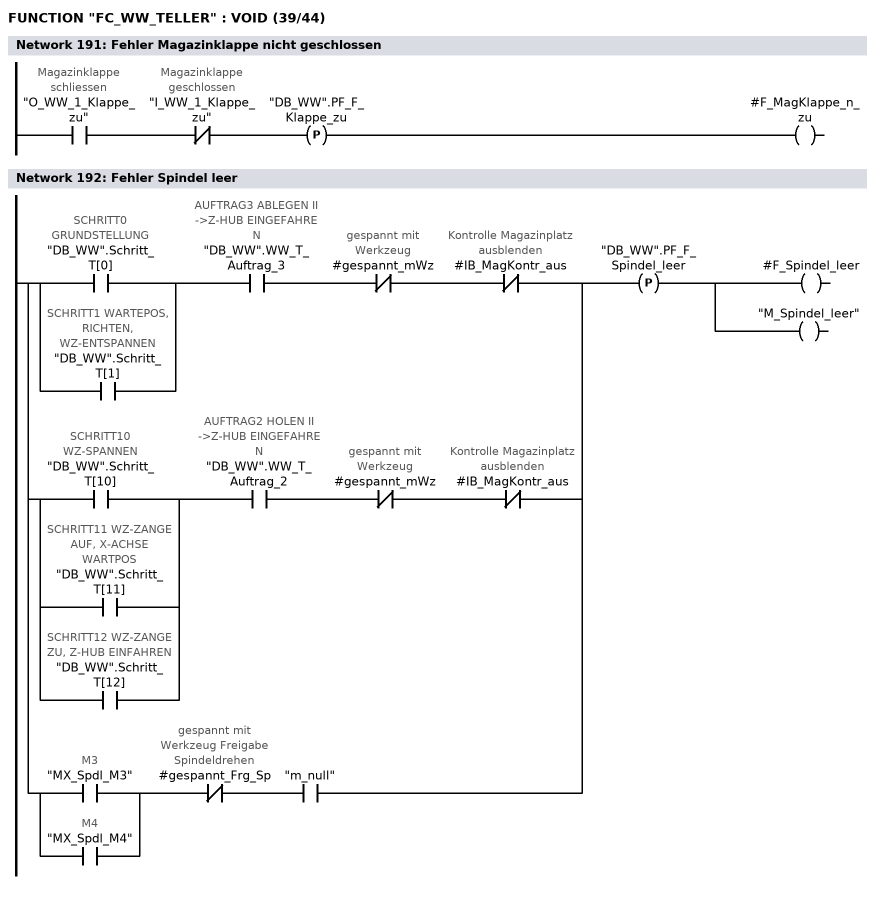

      U     "O_WW_1_Klappe_zu"; // Magazinklappe schliessen
      UN    "I_WW_1_Klappe_zu"; // Magazinklappe geschlossen
      FP    "DB_WW".PF_F_Klappe_zu;
      =     #F_MagKlappe_n_zu;

NETWORK
TITLE =Fehler Spindel leer

      U(    ;
      O     "DB_WW".Schritt_T[0]; // SCHRITT0 GRUNDSTELLUNG
      O     "DB_WW".Schritt_T[1]; // SCHRITT1 WARTEPOS, RICHTEN, WZ-ENTSPANNEN
      )     ;
      U     "DB_WW".WW_T_Auftrag_3; // AUFTRAG3 ABLEGEN II ->Z-HUB EINGEFAHREN
      UN    #gespannt_mWz; // gespannt mit Werkzeug
      UN    #IB_MagKontr_aus; // Kontrolle Magazinplatz ausblenden
      O     ;
      U(    ;
      O     "DB_WW".Schritt_T[10]; // SCHRITT10 WZ-SPANNEN
      O     "DB_WW".Schritt_T[11]; // SCHRITT11 WZ-ZANGE AUF, X-ACHSE WARTPOS
      O     "DB_WW".Schritt_T[12]; // SCHRITT12 WZ-ZANGE ZU, Z-HUB EINFAHREN
      )     ;
      U     "DB_WW".WW_T_Auftrag_2; // AUFTRAG2 HOLEN II ->Z-HUB EINGEFAHREN
      UN    #gespannt_mWz; // gespannt mit Werkzeug
      UN    #IB_MagKontr_aus; // Kontrolle Magazinplatz ausblenden
      O     ;
      U(    ;
      O     "MX_Spdl_M3"; //M3
      O     "MX_Spdl_M4"; //M4
      )     ;
      UN    #gespannt_Frg_Sp; // gespannt mit Werkzeug Freigabe Spindeldrehen
      U     "m_null";
      FP    "DB_WW".PF_F_Spindel_leer;
      =     #F_Spindel_leer;
      =     "M_Spindel_leer";
//      =     "DB_FEHLERMELDUNG".Spi_VS_Halt._700152_WZW_Nicht_Erlaub

NETWORK
TITLE =gespeicherte Fehlermeldungen löschen
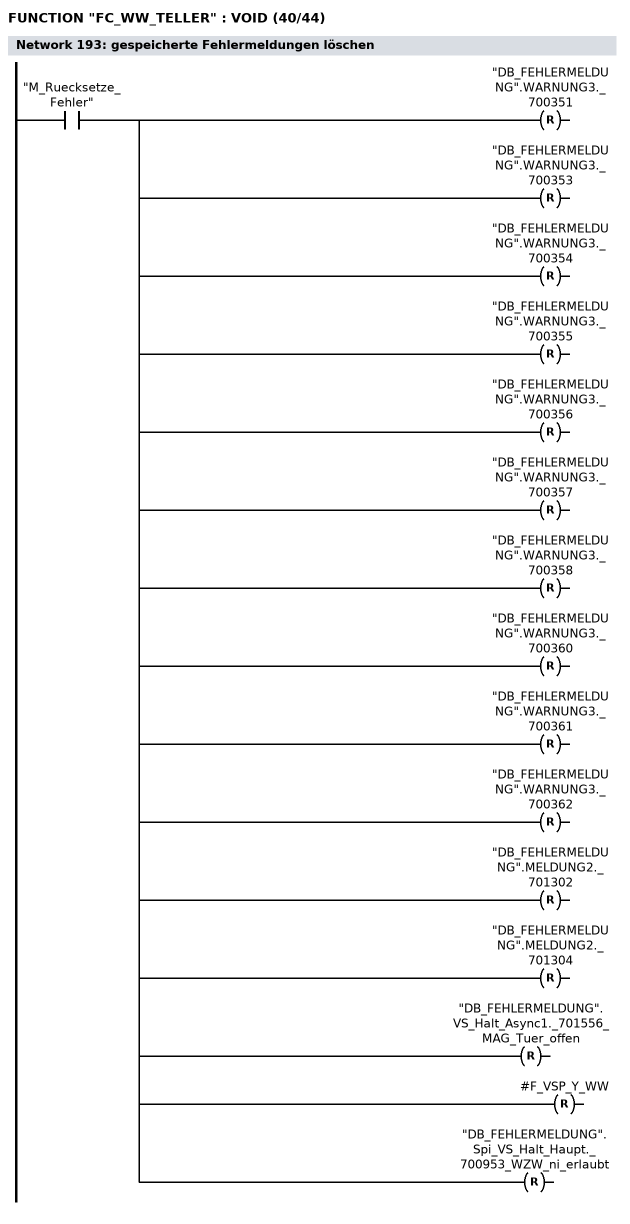

      U     "M_Ruecksetze_Fehler";
      R     "DB_FEHLERMELDUNG".WARNUNG3._700351;
      R     "DB_FEHLERMELDUNG".WARNUNG3._700353;
      R     "DB_FEHLERMELDUNG".WARNUNG3._700354;
      R     "DB_FEHLERMELDUNG".WARNUNG3._700355;
      R     "DB_FEHLERMELDUNG".WARNUNG3._700356;
      R     "DB_FEHLERMELDUNG".WARNUNG3._700357;
      R     "DB_FEHLERMELDUNG".WARNUNG3._700358;
      R     "DB_FEHLERMELDUNG".WARNUNG3._700360;
      R     "DB_FEHLERMELDUNG".WARNUNG3._700361;
      R     "DB_FEHLERMELDUNG".WARNUNG3._700362;
      R     "DB_FEHLERMELDUNG".MELDUNG2._701302;
      R     "DB_FEHLERMELDUNG".MELDUNG2._701304;

      R     "DB_FEHLERMELDUNG".VS_Halt_Async1._701556_MAG_Tuer_offen;
      R     #F_VSP_Y_WW;
      R     "DB_FEHLERMELDUNG".Spi_VS_Halt_Haupt._700953_WZW_ni_erlaubt;
NETWORK
TITLE =WZW nicht erlaubt
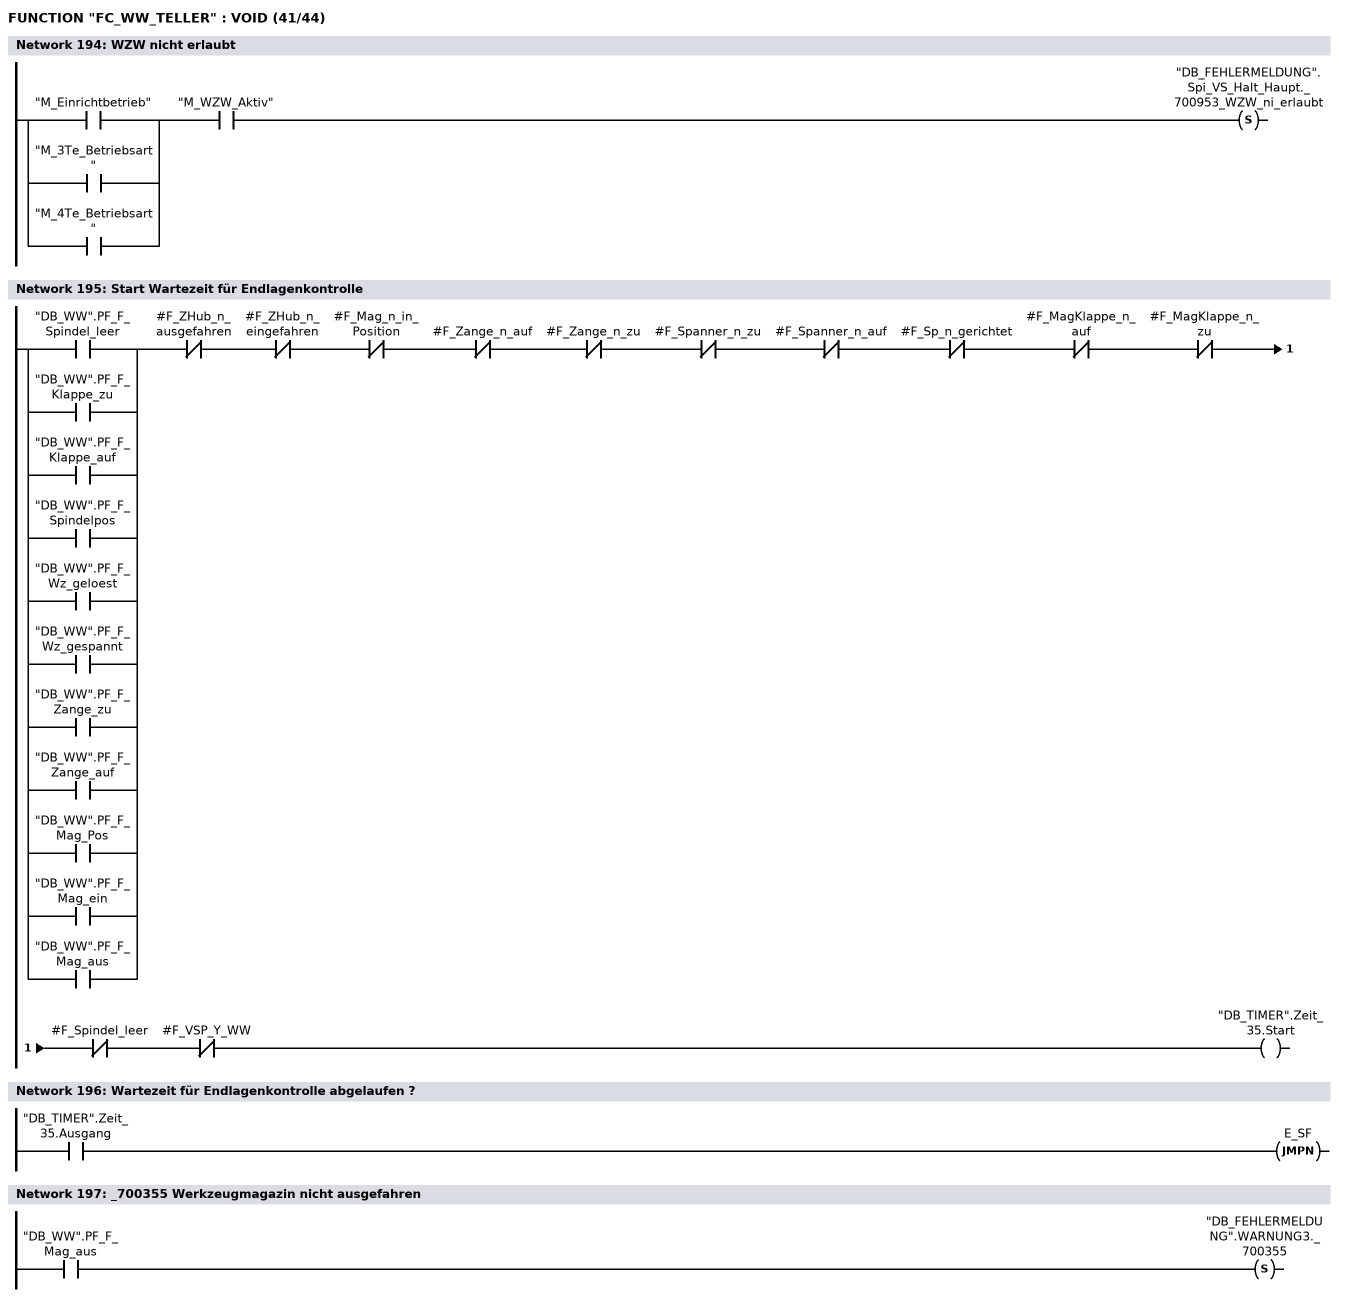

      U(    ;
      O     "M_Einrichtbetrieb";
      O     "M_3Te_Betriebsart";
      O     "M_4Te_Betriebsart";
      )     ;
      U     "M_WZW_Aktiv";
      S     "DB_FEHLERMELDUNG".Spi_VS_Halt_Haupt._700953_WZW_ni_erlaubt;
NETWORK
TITLE =Start Wartezeit für Endlagenkontrolle

      U(    ;
      O     "DB_WW".PF_F_Spindel_leer;
      O     "DB_WW".PF_F_Klappe_zu;
      O     "DB_WW".PF_F_Klappe_auf;
      O     "DB_WW".PF_F_Spindelpos;
      O     "DB_WW".PF_F_Wz_geloest;
      O     "DB_WW".PF_F_Wz_gespannt;
      O     "DB_WW".PF_F_Zange_zu;
      O     "DB_WW".PF_F_Zange_auf;
      O     "DB_WW".PF_F_Mag_Pos;
      O     "DB_WW".PF_F_Mag_ein;
      O     "DB_WW".PF_F_Mag_aus;
      )     ;
      UN    #F_ZHub_n_ausgefahren;
      UN    #F_ZHub_n_eingefahren;
      UN    #F_Mag_n_in_Position;
      UN    #F_Zange_n_auf;
      UN    #F_Zange_n_zu;
      UN    #F_Spanner_n_zu;
      UN    #F_Spanner_n_auf;
      UN    #F_Sp_n_gerichtet;
      UN    #F_MagKlappe_n_auf;
      UN    #F_MagKlappe_n_zu;
      UN    #F_Spindel_leer;
      UN    #F_VSP_Y_WW;

      =     "DB_TIMER".Zeit_35.Start;
NETWORK
TITLE =Wartezeit für Endlagenkontrolle abgelaufen ?

      U     "DB_TIMER".Zeit_35.Ausgang;
      SPBN  E_SF;

NETWORK
TITLE =_700355 Werkzeugmagazin nicht ausgefahren

      U     "DB_WW".PF_F_Mag_aus;
      S     "DB_FEHLERMELDUNG".WARNUNG3._700355;

NETWORK
TITLE =_700356 Werkzeugmagazin nicht eingefahren
